MoveL Offs(p0,431.3,226.6, 0), v100, z5, tool0;
MoveL Offs(p0,430.26560000000006,226.81200000000004, 0), v100, z5, tool0;
MoveL Offs(p0,429.7934,226.93749999999994, 0), v100, z5, tool0;
MoveL Offs(p0,429.36080000000004,227.07200000000003, 0), v100, z5, tool0;
MoveL Offs(p0,428.975,227.2125, 0), v100, z5, tool0;
MoveL Offs(p0,428.6432,227.356, 0), v100, z5, tool0;
MoveL Offs(p0,428.37260000000003,227.49949999999998, 0), v100, z5, tool0;
MoveL Offs(p0,428.1704,227.64000000000001, 0), v100, z5, tool0;
MoveL Offs(p0,428.04380000000003,227.77450000000005, 0), v100, z5, tool0;
MoveL Offs(p0,428.0,227.9, 0), v100, z5, tool0;
MoveL Offs(p0,427.0009999999999,228.11059999999998, 0), v100, z5, tool0;
MoveL Offs(p0,426.27200000000005,228.15120000000002, 0), v100, z5, tool0;
MoveL Offs(p0,425.375,228.175, 0), v100, z5, tool0;
MoveL Offs(p0,424.3280000000001,228.1808, 0), v100, z5, tool0;
MoveL Offs(p0,423.149,228.1674, 0), v100, z5, tool0;
MoveL Offs(p0,421.85600000000005,228.13360000000003, 0), v100, z5, tool0;
MoveL Offs(p0,410.99179999999996,228.3078, 0), v100, z5, tool0;
MoveL Offs(p0,411.1,228.5, 0), v100, z5, tool0;
MoveL Offs(p0,411.9424000000001,228.8344000000001, 0), v100, z5, tool0;
MoveL Offs(p0,412.7326,228.9806, 0), v100, z5, tool0;
MoveL Offs(p0,413.73519999999996,229.1112, 0), v100, z5, tool0;
MoveL Offs(p0,414.925,229.225, 0), v100, z5, tool0;
MoveL Offs(p0,416.2768,229.32080000000002, 0), v100, z5, tool0;
MoveL Offs(p0,417.76540000000006,229.3974, 0), v100, z5, tool0;
MoveL Offs(p0,419.3656,229.4536, 0), v100, z5, tool0;
MoveL Offs(p0,421.0522000000001,229.4882, 0), v100, z5, tool0;
MoveL Offs(p0,422.8,229.5, 0), v100, z5, tool0;
MoveL Offs(p0,431.6752,229.20240000000004, 0), v100, z5, tool0;
MoveL Offs(p0,433.1875,228.9375, 0), v100, z5, tool0;
MoveL Offs(p0,434.63680000000005,228.5496, 0), v100, z5, tool0;
MoveL Offs(p0,436.13289999999995,228.01530000000002, 0), v100, z5, tool0;
MoveL Offs(p0,437.7856,227.3112, 0), v100, z5, tool0;
MoveL Offs(p0,439.70470000000006,226.4139, 0), v100, z5, tool0;
MoveL Offs(p0,442.0,225.3, 0), v100, z5, tool0;
MoveL Offs(p0,448.8923,221.3112, 0), v100, z5, tool0;
MoveL Offs(p0,454.77840000000015,216.69360000000006, 0), v100, z5, tool0;
MoveL Offs(p0,459.6121,211.5804, 0), v100, z5, tool0;
MoveL Offs(p0,463.34720000000004,206.1048, 0), v100, z5, tool0;
MoveL Offs(p0,465.9375,200.4, 0), v100, z5, tool0;
MoveL Offs(p0,467.33680000000004,194.5992, 0), v100, z5, tool0;
MoveL Offs(p0,467.49889999999994,188.8356, 0), v100, z5, tool0;
MoveL Offs(p0,466.3776,183.2424, 0), v100, z5, tool0;
MoveL Offs(p0,463.9267,177.9528, 0), v100, z5, tool0;
MoveL Offs(p0,460.1,173.1, 0), v100, z5, tool0;
MoveL Offs(p0,458.00750000000005,171.084, 0), v100, z5, tool0;
MoveL Offs(p0,455.96000000000004,169.34400000000005, 0), v100, z5, tool0;
MoveL Offs(p0,453.9125,167.86200000000002, 0), v100, z5, tool0;
MoveL Offs(p0,451.82000000000005,166.62000000000003, 0), v100, z5, tool0;
MoveL Offs(p0,449.6375,165.6, 0), v100, z5, tool0;
MoveL Offs(p0,447.32,164.784, 0), v100, z5, tool0;
MoveL Offs(p0,444.82250000000005,164.154, 0), v100, z5, tool0;
MoveL Offs(p0,442.1,163.692, 0), v100, z5, tool0;
MoveL Offs(p0,439.10749999999996,163.38, 0), v100, z5, tool0;
MoveL Offs(p0,435.8,163.2, 0), v100, z5, tool0;
MoveL Offs(p0,425.2664,163.5024, 0), v100, z5, tool0;
MoveL Offs(p0,423.8902,163.76069999999999, 0), v100, z5, tool0;
MoveL Offs(p0,422.50079999999997,164.0928, 0), v100, z5, tool0;
MoveL Offs(p0,421.0526,164.50410000000002, 0), v100, z5, tool0;
MoveL Offs(p0,419.5,165.0, 0), v100, z5, tool0;
MoveL Offs(p0,418.4228,165.3736, 0), v100, z5, tool0;
MoveL Offs(p0,417.36240000000015,165.76880000000003, 0), v100, z5, tool0;
MoveL Offs(p0,416.3356,166.1772, 0), v100, z5, tool0;
MoveL Offs(p0,415.3592,166.59040000000002, 0), v100, z5, tool0;
MoveL Offs(p0,414.45,167.0, 0), v100, z5, tool0;
MoveL Offs(p0,413.62479999999994,167.3976, 0), v100, z5, tool0;
MoveL Offs(p0,412.9004,167.7748, 0), v100, z5, tool0;
MoveL Offs(p0,412.2936000000001,168.12320000000003, 0), v100, z5, tool0;
MoveL Offs(p0,411.82120000000003,168.4344, 0), v100, z5, tool0;
MoveL Offs(p0,411.5,168.7, 0), v100, z5, tool0;
MoveL Offs(p0,411.22180000000014,168.9393, 0), v100, z5, tool0;
MoveL Offs(p0,410.9304000000001,169.17440000000005, 0), v100, z5, tool0;
MoveL Offs(p0,410.63059999999996,169.4011, 0), v100, z5, tool0;
MoveL Offs(p0,410.3272,169.61520000000002, 0), v100, z5, tool0;
MoveL Offs(p0,410.025,169.8125, 0), v100, z5, tool0;
MoveL Offs(p0,409.72880000000004,169.9888, 0), v100, z5, tool0;
MoveL Offs(p0,409.4434,170.13989999999998, 0), v100, z5, tool0;
MoveL Offs(p0,409.17359999999996,170.2616, 0), v100, z5, tool0;
MoveL Offs(p0,408.92420000000004,170.3497, 0), v100, z5, tool0;
MoveL Offs(p0,408.7,170.4, 0), v100, z5, tool0;
MoveL Offs(p0,407.1136000000001,170.85280000000006, 0), v100, z5, tool0;
MoveL Offs(p0,406.3384,171.20819999999998, 0), v100, z5, tool0;
MoveL Offs(p0,405.6088000000001,171.62240000000003, 0), v100, z5, tool0;
MoveL Offs(p0,404.95,172.075, 0), v100, z5, tool0;
MoveL Offs(p0,404.3872,172.54559999999998, 0), v100, z5, tool0;
MoveL Offs(p0,403.9456,173.0138, 0), v100, z5, tool0;
MoveL Offs(p0,403.65040000000005,173.4592, 0), v100, z5, tool0;
MoveL Offs(p0,403.52680000000004,173.8614, 0), v100, z5, tool0;
MoveL Offs(p0,403.6,174.2, 0), v100, z5, tool0;
MoveL Offs(p0,403.8223,174.67069999999998, 0), v100, z5, tool0;
MoveL Offs(p0,403.83360000000005,174.75840000000002, 0), v100, z5, tool0;
MoveL Offs(p0,403.8125,174.8125, 0), v100, z5, tool0;
MoveL Offs(p0,403.3921,174.7049, 0), v100, z5, tool0;
MoveL Offs(p0,403.2,174.6, 0), v100, z5, tool0;
MoveL Offs(p0,401.24240000000015,175.26400000000007, 0), v100, z5, tool0;
MoveL Offs(p0,399.7251,176.45850000000002, 0), v100, z5, tool0;
MoveL Offs(p0,397.9552,178.11200000000002, 0), v100, z5, tool0;
MoveL Offs(p0,396.0125,180.1375, 0), v100, z5, tool0;
MoveL Offs(p0,393.9768,182.448, 0), v100, z5, tool0;
MoveL Offs(p0,391.9279,184.9565, 0), v100, z5, tool0;
MoveL Offs(p0,389.94560000000007,187.57600000000002, 0), v100, z5, tool0;
MoveL Offs(p0,388.10970000000003,190.2195, 0), v100, z5, tool0;
MoveL Offs(p0,386.5,192.8, 0), v100, z5, tool0;
MoveL Offs(p0,385.22280000000006,195.07940000000002, 0), v100, z5, tool0;
MoveL Offs(p0,383.87840000000017,197.65520000000004, 0), v100, z5, tool0;
MoveL Offs(p0,382.5076,200.43380000000002, 0), v100, z5, tool0;
MoveL Offs(p0,381.1512,203.32160000000002, 0), v100, z5, tool0;
MoveL Offs(p0,379.85,206.225, 0), v100, z5, tool0;
MoveL Offs(p0,378.6448,209.05040000000002, 0), v100, z5, tool0;
MoveL Offs(p0,377.57640000000004,211.7042, 0), v100, z5, tool0;
MoveL Offs(p0,376.6856,214.09279999999998, 0), v100, z5, tool0;
MoveL Offs(p0,376.0132,216.1226, 0), v100, z5, tool0;
MoveL Offs(p0,375.6,217.7, 0), v100, z5, tool0;
MoveL Offs(p0,375.1392,219.68720000000002, 0), v100, z5, tool0;
MoveL Offs(p0,374.49360000000013,221.77760000000006, 0), v100, z5, tool0;
MoveL Offs(p0,373.6884,223.92439999999996, 0), v100, z5, tool0;
MoveL Offs(p0,372.7488000000001,226.0808, 0), v100, z5, tool0;
MoveL Offs(p0,371.7,228.2, 0), v100, z5, tool0;
MoveL Offs(p0,370.56719999999996,230.2352, 0), v100, z5, tool0;
MoveL Offs(p0,369.3756,232.13959999999997, 0), v100, z5, tool0;
MoveL Offs(p0,368.15040000000005,233.86640000000003, 0), v100, z5, tool0;
MoveL Offs(p0,366.9168,235.36880000000002, 0), v100, z5, tool0;
MoveL Offs(p0,365.7,236.6, 0), v100, z5, tool0;
MoveL Offs(p0,363.6746,238.30100000000002, 0), v100, z5, tool0;
MoveL Offs(p0,361.6168000000001,239.74400000000009, 0), v100, z5, tool0;
MoveL Offs(p0,359.52419999999995,240.929, 0), v100, z5, tool0;
MoveL Offs(p0,357.3944,241.85600000000005, 0), v100, z5, tool0;
MoveL Offs(p0,355.225,242.525, 0), v100, z5, tool0;
MoveL Offs(p0,353.0136,242.93599999999998, 0), v100, z5, tool0;
MoveL Offs(p0,350.75780000000003,243.08900000000003, 0), v100, z5, tool0;
MoveL Offs(p0,348.45520000000005,242.984, 0), v100, z5, tool0;
MoveL Offs(p0,346.1034,242.621, 0), v100, z5, tool0;
MoveL Offs(p0,343.7,242.0, 0), v100, z5, tool0;
MoveL Offs(p0,338.0,240.2, 0), v100, z5, tool0;
MoveL Offs(p0,338.0,243.0, 0), v100, z5, tool0;
MoveL Offs(p0,338.43520000000007,245.01520000000005, 0), v100, z5, tool0;
MoveL Offs(p0,339.0098,245.79179999999997, 0), v100, z5, tool0;
MoveL Offs(p0,339.84959999999995,246.42560000000003, 0), v100, z5, tool0;
MoveL Offs(p0,340.975,246.925, 0), v100, z5, tool0;
MoveL Offs(p0,342.40639999999996,247.2984, 0), v100, z5, tool0;
MoveL Offs(p0,344.1642,247.55419999999998, 0), v100, z5, tool0;
MoveL Offs(p0,346.2688,247.70080000000002, 0), v100, z5, tool0;
MoveL Offs(p0,348.7406,247.7466, 0), v100, z5, tool0;
MoveL Offs(p0,351.6,247.7, 0), v100, z5, tool0;
MoveL Offs(p0,355.35920000000004,247.4872000000001, 0), v100, z5, tool0;
MoveL Offs(p0,356.85779999999994,247.3328, 0), v100, z5, tool0;
MoveL Offs(p0,358.17760000000004,247.1256, 0), v100, z5, tool0;
MoveL Offs(p0,359.375,246.85, 0), v100, z5, tool0;
MoveL Offs(p0,360.50640000000004,246.4904, 0), v100, z5, tool0;
MoveL Offs(p0,361.6282,246.03119999999998, 0), v100, z5, tool0;
MoveL Offs(p0,362.79679999999996,245.45680000000002, 0), v100, z5, tool0;
MoveL Offs(p0,364.0686,244.7516, 0), v100, z5, tool0;
MoveL Offs(p0,365.5,243.9, 0), v100, z5, tool0;
MoveL Offs(p0,365.5,243.9, 0), v100, z5, tool0;
MoveJ Offs(p0,333.7,242.7, 10), v100, z1, tool0;
MoveL Offs(p0,333.3992,241.44880000000003, 0), v100, z5, tool0;
MoveL Offs(p0,333.2194,241.6821, 0), v100, z5, tool0;
MoveL Offs(p0,333.0,242.0, 0), v100, z5, tool0;
MoveL Offs(p0,332.6946000000001,242.54360000000003, 0), v100, z5, tool0;
MoveL Offs(p0,332.44080000000014,243.13280000000003, 0), v100, z5, tool0;
MoveL Offs(p0,332.2422,243.7352, 0), v100, z5, tool0;
MoveL Offs(p0,332.10240000000005,244.31840000000003, 0), v100, z5, tool0;
MoveL Offs(p0,332.025,244.85, 0), v100, z5, tool0;
MoveL Offs(p0,332.0136,245.29759999999996, 0), v100, z5, tool0;
MoveL Offs(p0,332.0718,245.6288, 0), v100, z5, tool0;
MoveL Offs(p0,332.20320000000004,245.8112, 0), v100, z5, tool0;
MoveL Offs(p0,332.4114,245.81239999999997, 0), v100, z5, tool0;
MoveL Offs(p0,332.7,245.6, 0), v100, z5, tool0;
MoveL Offs(p0,332.9384000000001,245.29840000000007, 0), v100, z5, tool0;
MoveL Offs(p0,333.0546,245.06809999999996, 0), v100, z5, tool0;
MoveL Offs(p0,333.16720000000004,244.79520000000002, 0), v100, z5, tool0;
MoveL Offs(p0,333.275,244.4875, 0), v100, z5, tool0;
MoveL Offs(p0,333.3768,244.15279999999998, 0), v100, z5, tool0;
MoveL Offs(p0,333.4714,243.7989, 0), v100, z5, tool0;
MoveL Offs(p0,333.5576,243.4336, 0), v100, z5, tool0;
MoveL Offs(p0,333.6342,243.0647, 0), v100, z5, tool0;
MoveL Offs(p0,333.7,242.7, 0), v100, z5, tool0;
MoveL Offs(p0,333.7,242.7, 0), v100, z5, tool0;
MoveJ Offs(p0,201.3,238.9, 10), v100, z1, tool0;
MoveL Offs(p0,202.17000000000002,238.3953, 0), v100, z5, tool0;
MoveL Offs(p0,203.13600000000005,237.74240000000003, 0), v100, z5, tool0;
MoveL Offs(p0,204.16199999999998,236.9731, 0), v100, z5, tool0;
MoveL Offs(p0,205.212,236.11920000000003, 0), v100, z5, tool0;
MoveL Offs(p0,206.25,235.2125, 0), v100, z5, tool0;
MoveL Offs(p0,207.24,234.2848, 0), v100, z5, tool0;
MoveL Offs(p0,208.14600000000002,233.36790000000002, 0), v100, z5, tool0;
MoveL Offs(p0,208.93200000000002,232.49360000000001, 0), v100, z5, tool0;
MoveL Offs(p0,209.56199999999998,231.69369999999998, 0), v100, z5, tool0;
MoveL Offs(p0,210.0,231.0, 0), v100, z5, tool0;
MoveL Offs(p0,209.68800000000002,229.92960000000002, 0), v100, z5, tool0;
MoveL Offs(p0,209.1375,229.8, 0), v100, z5, tool0;
MoveL Offs(p0,208.344,229.71840000000003, 0), v100, z5, tool0;
MoveL Offs(p0,207.2805,229.6812, 0), v100, z5, tool0;
MoveL Offs(p0,205.92000000000002,229.6848, 0), v100, z5, tool0;
MoveL Offs(p0,204.2355,229.72560000000004, 0), v100, z5, tool0;
MoveL Offs(p0,202.2,229.8, 0), v100, z5, tool0;
MoveL Offs(p0,188.76839999999999,229.2276, 0), v100, z5, tool0;
MoveL Offs(p0,183.70880000000002,228.5232, 0), v100, z5, tool0;
MoveL Offs(p0,178.3,227.55, 0), v100, z5, tool0;
MoveL Offs(p0,172.50719999999995,226.30079999999998, 0), v100, z5, tool0;
MoveL Offs(p0,166.2956,224.76839999999999, 0), v100, z5, tool0;
MoveL Offs(p0,159.6304,222.9456, 0), v100, z5, tool0;
MoveL Offs(p0,152.4768,220.8252, 0), v100, z5, tool0;
MoveL Offs(p0,144.8,218.4, 0), v100, z5, tool0;
MoveL Offs(p0,137.62550000000002,215.98860000000005, 0), v100, z5, tool0;
MoveL Offs(p0,130.28000000000003,213.31680000000006, 0), v100, z5, tool0;
MoveL Offs(p0,122.97050000000002,210.47819999999996, 0), v100, z5, tool0;
MoveL Offs(p0,115.90400000000002,207.56640000000002, 0), v100, z5, tool0;
MoveL Offs(p0,109.2875,204.675, 0), v100, z5, tool0;
MoveL Offs(p0,103.328,201.8976, 0), v100, z5, tool0;
MoveL Offs(p0,98.23249999999999,199.3278, 0), v100, z5, tool0;
MoveL Offs(p0,94.20800000000001,197.0592, 0), v100, z5, tool0;
MoveL Offs(p0,91.4615,195.18540000000002, 0), v100, z5, tool0;
MoveL Offs(p0,90.2,193.8, 0), v100, z5, tool0;
MoveL Offs(p0,89.98890000000002,193.48160000000001, 0), v100, z5, tool0;
MoveL Offs(p0,89.67520000000002,193.24480000000003, 0), v100, z5, tool0;
MoveL Offs(p0,89.2883,193.0872, 0), v100, z5, tool0;
MoveL Offs(p0,88.85760000000002,193.0064, 0), v100, z5, tool0;
MoveL Offs(p0,88.4125,193.0, 0), v100, z5, tool0;
MoveL Offs(p0,87.9824,193.0656, 0), v100, z5, tool0;
MoveL Offs(p0,87.5967,193.2008, 0), v100, z5, tool0;
MoveL Offs(p0,87.2848,193.40320000000003, 0), v100, z5, tool0;
MoveL Offs(p0,87.0,194.0, 0), v100, z5, tool0;
MoveL Offs(p0,86.7376,194.6112, 0), v100, z5, tool0;
MoveL Offs(p0,86.6,194.725, 0), v100, z5, tool0;
MoveL Offs(p0,86.43839999999999,194.82080000000002, 0), v100, z5, tool0;
MoveL Offs(p0,86.2552,194.8974, 0), v100, z5, tool0;
MoveL Offs(p0,86.0528,194.9536, 0), v100, z5, tool0;
MoveL Offs(p0,85.8336,194.9882, 0), v100, z5, tool0;
MoveL Offs(p0,85.6,195.0, 0), v100, z5, tool0;
MoveL Offs(p0,84.32000000000002,195.36960000000002, 0), v100, z5, tool0;
MoveL Offs(p0,83.8945,195.78839999999997, 0), v100, z5, tool0;
MoveL Offs(p0,83.61600000000001,196.3248, 0), v100, z5, tool0;
MoveL Offs(p0,83.4875,196.95, 0), v100, z5, tool0;
MoveL Offs(p0,83.51200000000001,197.6352, 0), v100, z5, tool0;
MoveL Offs(p0,83.6925,198.35160000000002, 0), v100, z5, tool0;
MoveL Offs(p0,84.03200000000001,199.0704, 0), v100, z5, tool0;
MoveL Offs(p0,84.5335,199.76280000000003, 0), v100, z5, tool0;
MoveL Offs(p0,85.2,200.4, 0), v100, z5, tool0;
MoveL Offs(p0,86.3957,201.25300000000001, 0), v100, z5, tool0;
MoveL Offs(p0,88.03360000000004,202.26800000000006, 0), v100, z5, tool0;
MoveL Offs(p0,89.9799,203.379, 0), v100, z5, tool0;
MoveL Offs(p0,92.10080000000002,204.52000000000004, 0), v100, z5, tool0;
MoveL Offs(p0,94.2625,205.625, 0), v100, z5, tool0;
MoveL Offs(p0,96.3312,206.62800000000001, 0), v100, z5, tool0;
MoveL Offs(p0,98.1731,207.46300000000002, 0), v100, z5, tool0;
MoveL Offs(p0,99.65440000000001,208.06400000000002, 0), v100, z5, tool0;
MoveL Offs(p0,100.6413,208.365, 0), v100, z5, tool0;
MoveL Offs(p0,101.0,208.3, 0), v100, z5, tool0;
MoveL Offs(p0,101.25,208.0375, 0), v100, z5, tool0;
MoveL Offs(p0,101.3456,208.09120000000001, 0), v100, z5, tool0;
MoveL Offs(p0,101.8,208.6, 0), v100, z5, tool0;
MoveL Offs(p0,102.76490000000001,209.33620000000005, 0), v100, z5, tool0;
MoveL Offs(p0,104.76720000000003,210.39760000000007, 0), v100, z5, tool0;
MoveL Offs(p0,107.5483,211.68339999999998, 0), v100, z5, tool0;
MoveL Offs(p0,110.84960000000001,213.09280000000004, 0), v100, z5, tool0;
MoveL Offs(p0,114.4125,214.525, 0), v100, z5, tool0;
MoveL Offs(p0,117.97840000000001,215.87920000000003, 0), v100, z5, tool0;
MoveL Offs(p0,121.28870000000002,217.05460000000002, 0), v100, z5, tool0;
MoveL Offs(p0,124.08480000000002,217.9504, 0), v100, z5, tool0;
MoveL Offs(p0,126.10810000000001,218.46580000000003, 0), v100, z5, tool0;
MoveL Offs(p0,127.1,218.5, 0), v100, z5, tool0;
MoveL Offs(p0,127.46960000000004,218.27120000000008, 0), v100, z5, tool0;
MoveL Offs(p0,127.61389999999999,218.20929999999998, 0), v100, z5, tool0;
MoveL Offs(p0,127.72880000000002,218.18159999999997, 0), v100, z5, tool0;
MoveL Offs(p0,127.8125,218.1875, 0), v100, z5, tool0;
MoveL Offs(p0,127.86319999999998,218.2264, 0), v100, z5, tool0;
MoveL Offs(p0,127.87910000000002,218.2977, 0), v100, z5, tool0;
MoveL Offs(p0,127.7,218.7, 0), v100, z5, tool0;
MoveL Offs(p0,128.13320000000002,219.17020000000002, 0), v100, z5, tool0;
MoveL Offs(p0,129.6896,220.0016000000001, 0), v100, z5, tool0;
MoveL Offs(p0,132.2144,221.13539999999998, 0), v100, z5, tool0;
MoveL Offs(p0,135.5528,222.51280000000003, 0), v100, z5, tool0;
MoveL Offs(p0,139.55,224.075, 0), v100, z5, tool0;
MoveL Offs(p0,144.05120000000002,225.7632, 0), v100, z5, tool0;
MoveL Offs(p0,148.9016,227.51859999999996, 0), v100, z5, tool0;
MoveL Offs(p0,153.9464,229.2824, 0), v100, z5, tool0;
MoveL Offs(p0,159.0308,230.9958, 0), v100, z5, tool0;
MoveL Offs(p0,164.0,232.6, 0), v100, z5, tool0;
MoveL Offs(p0,170.2905,234.5179, 0), v100, z5, tool0;
MoveL Offs(p0,175.92400000000006,236.13520000000008, 0), v100, z5, tool0;
MoveL Offs(p0,180.9335,237.45729999999998, 0), v100, z5, tool0;
MoveL Offs(p0,185.35200000000003,238.48960000000002, 0), v100, z5, tool0;
MoveL Offs(p0,189.2125,239.2375, 0), v100, z5, tool0;
MoveL Offs(p0,192.548,239.70639999999997, 0), v100, z5, tool0;
MoveL Offs(p0,195.3915,239.90169999999998, 0), v100, z5, tool0;
MoveL Offs(p0,197.776,239.82880000000006, 0), v100, z5, tool0;
MoveL Offs(p0,199.7345,239.4931, 0), v100, z5, tool0;
MoveL Offs(p0,201.3,238.9, 0), v100, z5, tool0;
MoveL Offs(p0,201.3,238.9, 0), v100, z5, tool0;
MoveJ Offs(p0,169.0,237.4, 10), v100, z1, tool0;
MoveL Offs(p0,168.7024,237.1728, 0), v100, z5, tool0;
MoveL Offs(p0,168.55,237.125, 0), v100, z5, tool0;
MoveL Offs(p0,168.37359999999998,237.08319999999998, 0), v100, z5, tool0;
MoveL Offs(p0,168.17680000000001,237.0486, 0), v100, z5, tool0;
MoveL Offs(p0,167.9632,237.0224, 0), v100, z5, tool0;
MoveL Offs(p0,167.7364,237.0058, 0), v100, z5, tool0;
MoveL Offs(p0,167.5,237.0, 0), v100, z5, tool0;
MoveL Offs(p0,166.45,237.275, 0), v100, z5, tool0;
MoveL Offs(p0,166.2976,237.3888, 0), v100, z5, tool0;
MoveL Offs(p0,166.1728,237.5194, 0), v100, z5, tool0;
MoveL Offs(p0,166.07920000000001,237.66559999999998, 0), v100, z5, tool0;
MoveL Offs(p0,166.0204,237.82620000000003, 0), v100, z5, tool0;
MoveL Offs(p0,166.0,238.0, 0), v100, z5, tool0;
MoveL Offs(p0,166.29760000000002,238.44320000000002, 0), v100, z5, tool0;
MoveL Offs(p0,166.45,238.5, 0), v100, z5, tool0;
MoveL Offs(p0,166.62640000000002,238.5328, 0), v100, z5, tool0;
MoveL Offs(p0,166.82319999999999,238.54039999999995, 0), v100, z5, tool0;
MoveL Offs(p0,167.03680000000003,238.52160000000003, 0), v100, z5, tool0;
MoveL Offs(p0,167.2636,238.4752, 0), v100, z5, tool0;
MoveL Offs(p0,167.5,238.4, 0), v100, z5, tool0;
MoveL Offs(p0,167.96320000000003,238.16160000000008, 0), v100, z5, tool0;
MoveL Offs(p0,168.17680000000001,238.04539999999997, 0), v100, z5, tool0;
MoveL Offs(p0,168.3736,237.93280000000004, 0), v100, z5, tool0;
MoveL Offs(p0,168.55,237.825, 0), v100, z5, tool0;
MoveL Offs(p0,168.7024,237.7232, 0), v100, z5, tool0;
MoveL Offs(p0,168.8272,237.6286, 0), v100, z5, tool0;
MoveL Offs(p0,168.9208,237.5424, 0), v100, z5, tool0;
MoveL Offs(p0,168.97960000000003,237.46580000000003, 0), v100, z5, tool0;
MoveL Offs(p0,169.0,237.4, 0), v100, z5, tool0;
MoveL Offs(p0,169.0,237.4, 0), v100, z5, tool0;
MoveJ Offs(p0,48.2,226.6, 10), v100, z1, tool0;
MoveL Offs(p0,51.083000000000006,225.5016, 0), v100, z5, tool0;
MoveL Offs(p0,53.55200000000001,224.12480000000005, 0), v100, z5, tool0;
MoveL Offs(p0,55.607000000000006,222.46719999999996, 0), v100, z5, tool0;
MoveL Offs(p0,57.248000000000005,220.52639999999997, 0), v100, z5, tool0;
MoveL Offs(p0,58.475,218.3, 0), v100, z5, tool0;
MoveL Offs(p0,59.28800000000001,215.7856, 0), v100, z5, tool0;
MoveL Offs(p0,59.687,212.9808, 0), v100, z5, tool0;
MoveL Offs(p0,59.672000000000004,209.88320000000004, 0), v100, z5, tool0;
MoveL Offs(p0,59.24300000000001,206.4904, 0), v100, z5, tool0;
MoveL Offs(p0,58.4,202.8, 0), v100, z5, tool0;
MoveL Offs(p0,58.19,201.4805, 0), v100, z5, tool0;
MoveL Offs(p0,58.16000000000001,201.28000000000003, 0), v100, z5, tool0;
MoveL Offs(p0,58.129999999999995,201.0855, 0), v100, z5, tool0;
MoveL Offs(p0,58.1,200.9, 0), v100, z5, tool0;
MoveL Offs(p0,57.8856,200.4568, 0), v100, z5, tool0;
MoveL Offs(p0,57.775,200.4, 0), v100, z5, tool0;
MoveL Offs(p0,57.64639999999999,200.36719999999997, 0), v100, z5, tool0;
MoveL Offs(p0,57.502199999999995,200.3596, 0), v100, z5, tool0;
MoveL Offs(p0,57.344800000000006,200.3784, 0), v100, z5, tool0;
MoveL Offs(p0,57.17660000000001,200.4248, 0), v100, z5, tool0;
MoveL Offs(p0,57.0,200.5, 0), v100, z5, tool0;
MoveL Offs(p0,56.4596,200.248, 0), v100, z5, tool0;
MoveL Offs(p0,56.47840000000001,200.06800000000004, 0), v100, z5, tool0;
MoveL Offs(p0,56.524800000000006,199.85200000000003, 0), v100, z5, tool0;
MoveL Offs(p0,56.6,199.6, 0), v100, z5, tool0;
MoveL Offs(p0,56.2193,196.98549999999997, 0), v100, z5, tool0;
MoveL Offs(p0,55.76160000000001,195.76000000000002, 0), v100, z5, tool0;
MoveL Offs(p0,55.1875,194.4625, 0), v100, z5, tool0;
MoveL Offs(p0,54.52639999999999,193.156, 0), v100, z5, tool0;
MoveL Offs(p0,53.8077,191.90350000000004, 0), v100, z5, tool0;
MoveL Offs(p0,53.06080000000001,190.76800000000003, 0), v100, z5, tool0;
MoveL Offs(p0,52.31510000000001,189.8125, 0), v100, z5, tool0;
MoveL Offs(p0,51.6,189.1, 0), v100, z5, tool0;
MoveL Offs(p0,51.2356,188.80980000000005, 0), v100, z5, tool0;
MoveL Offs(p0,50.916800000000016,188.60240000000005, 0), v100, z5, tool0;
MoveL Offs(p0,50.6352,188.4826, 0), v100, z5, tool0;
MoveL Offs(p0,50.382400000000004,188.45520000000002, 0), v100, z5, tool0;
MoveL Offs(p0,50.15,188.525, 0), v100, z5, tool0;
MoveL Offs(p0,49.92959999999999,188.6968, 0), v100, z5, tool0;
MoveL Offs(p0,49.491200000000006,189.36560000000003, 0), v100, z5, tool0;
MoveL Offs(p0,49.2564,189.8722, 0), v100, z5, tool0;
MoveL Offs(p0,49.0,190.5, 0), v100, z5, tool0;
MoveL Offs(p0,48.689600000000006,191.40240000000003, 0), v100, z5, tool0;
MoveL Offs(p0,48.5734,191.84459999999996, 0), v100, z5, tool0;
MoveL Offs(p0,48.4848,192.27120000000002, 0), v100, z5, tool0;
MoveL Offs(p0,48.425,192.675, 0), v100, z5, tool0;
MoveL Offs(p0,48.3952,193.04879999999997, 0), v100, z5, tool0;
MoveL Offs(p0,48.3966,193.38539999999998, 0), v100, z5, tool0;
MoveL Offs(p0,48.430400000000006,193.67760000000004, 0), v100, z5, tool0;
MoveL Offs(p0,48.4978,193.9182, 0), v100, z5, tool0;
MoveL Offs(p0,48.6,194.1, 0), v100, z5, tool0;
MoveL Offs(p0,48.3,194.8, 0), v100, z5, tool0;
MoveL Offs(p0,47.333600000000004,195.12640000000002, 0), v100, z5, tool0;
MoveL Offs(p0,46.975,195.3625, 0), v100, z5, tool0;
MoveL Offs(p0,46.5864,195.64960000000002, 0), v100, z5, tool0;
MoveL Offs(p0,46.176199999999994,195.98229999999998, 0), v100, z5, tool0;
MoveL Offs(p0,45.7528,196.35520000000002, 0), v100, z5, tool0;
MoveL Offs(p0,45.3246,196.7629, 0), v100, z5, tool0;
MoveL Offs(p0,44.9,197.2, 0), v100, z5, tool0;
MoveL Offs(p0,43.92960000000001,198.06340000000003, 0), v100, z5, tool0;
MoveL Offs(p0,42.82480000000001,198.85120000000006, 0), v100, z5, tool0;
MoveL Offs(p0,41.59519999999999,199.5598, 0), v100, z5, tool0;
MoveL Offs(p0,40.2504,200.1856, 0), v100, z5, tool0;
MoveL Offs(p0,38.8,200.725, 0), v100, z5, tool0;
MoveL Offs(p0,37.2536,201.1744, 0), v100, z5, tool0;
MoveL Offs(p0,35.620799999999996,201.53019999999998, 0), v100, z5, tool0;
MoveL Offs(p0,33.911199999999994,201.7888, 0), v100, z5, tool0;
MoveL Offs(p0,32.13440000000001,201.94660000000002, 0), v100, z5, tool0;
MoveL Offs(p0,30.3,202.0, 0), v100, z5, tool0;
MoveL Offs(p0,26.2,202.0, 0), v100, z5, tool0;
MoveL Offs(p0,28.1,208.3, 0), v100, z5, tool0;
MoveL Offs(p0,28.396200000000004,209.35530000000003, 0), v100, z5, tool0;
MoveL Offs(p0,28.681600000000003,210.46640000000008, 0), v100, z5, tool0;
MoveL Offs(p0,28.9514,211.6111, 0), v100, z5, tool0;
MoveL Offs(p0,29.200799999999997,212.7672, 0), v100, z5, tool0;
MoveL Offs(p0,29.425,213.9125, 0), v100, z5, tool0;
MoveL Offs(p0,29.6192,215.0248, 0), v100, z5, tool0;
MoveL Offs(p0,29.7786,216.0819, 0), v100, z5, tool0;
MoveL Offs(p0,29.898400000000002,217.0616, 0), v100, z5, tool0;
MoveL Offs(p0,29.9738,217.9417, 0), v100, z5, tool0;
MoveL Offs(p0,30.0,218.7, 0), v100, z5, tool0;
MoveL Offs(p0,30.352000000000004,222.07280000000006, 0), v100, z5, tool0;
MoveL Offs(p0,30.6125,222.6625, 0), v100, z5, tool0;
MoveL Offs(p0,30.972,223.2072, 0), v100, z5, tool0;
MoveL Offs(p0,31.4455,223.73509999999996, 0), v100, z5, tool0;
MoveL Offs(p0,32.048,224.27439999999996, 0), v100, z5, tool0;
MoveL Offs(p0,32.7945,224.85330000000005, 0), v100, z5, tool0;
MoveL Offs(p0,33.7,225.5, 0), v100, z5, tool0;
MoveL Offs(p0,34.96730000000001,226.26520000000005, 0), v100, z5, tool0;
MoveL Offs(p0,36.20640000000001,226.88160000000008, 0), v100, z5, tool0;
MoveL Offs(p0,37.4431,227.35040000000004, 0), v100, z5, tool0;
MoveL Offs(p0,38.7032,227.6728, 0), v100, z5, tool0;
MoveL Offs(p0,40.0125,227.85, 0), v100, z5, tool0;
MoveL Offs(p0,41.3968,227.8832, 0), v100, z5, tool0;
MoveL Offs(p0,42.881899999999995,227.7736, 0), v100, z5, tool0;
MoveL Offs(p0,44.4936,227.5224, 0), v100, z5, tool0;
MoveL Offs(p0,46.2577,227.1308, 0), v100, z5, tool0;
MoveL Offs(p0,48.2,226.6, 0), v100, z5, tool0;
MoveL Offs(p0,48.2,226.6, 0), v100, z5, tool0;
MoveJ Offs(p0,209.9,227.4, 10), v100, z1, tool0;
MoveL Offs(p0,211.07630000000003,227.07440000000005, 0), v100, z5, tool0;
MoveL Offs(p0,211.96640000000002,226.64320000000006, 0), v100, z5, tool0;
MoveL Offs(p0,212.5721,226.11479999999997, 0), v100, z5, tool0;
MoveL Offs(p0,212.89520000000002,225.4976, 0), v100, z5, tool0;
MoveL Offs(p0,212.9375,224.8, 0), v100, z5, tool0;
MoveL Offs(p0,212.7008,224.03040000000001, 0), v100, z5, tool0;
MoveL Offs(p0,212.18689999999998,223.19719999999998, 0), v100, z5, tool0;
MoveL Offs(p0,211.3976,222.30880000000002, 0), v100, z5, tool0;
MoveL Offs(p0,210.33469999999997,221.37359999999998, 0), v100, z5, tool0;
MoveL Offs(p0,209.0,220.4, 0), v100, z5, tool0;
MoveL Offs(p0,207.7799,219.58109999999996, 0), v100, z5, tool0;
MoveL Offs(p0,206.8112,218.90080000000006, 0), v100, z5, tool0;
MoveL Offs(p0,206.08129999999997,218.32369999999997, 0), v100, z5, tool0;
MoveL Offs(p0,205.57760000000002,217.81440000000003, 0), v100, z5, tool0;
MoveL Offs(p0,205.2875,217.3375, 0), v100, z5, tool0;
MoveL Offs(p0,205.1984,216.8576, 0), v100, z5, tool0;
MoveL Offs(p0,205.2977,216.3393, 0), v100, z5, tool0;
MoveL Offs(p0,205.5728,215.74720000000002, 0), v100, z5, tool0;
MoveL Offs(p0,206.01110000000003,215.0459, 0), v100, z5, tool0;
MoveL Offs(p0,206.6,214.2, 0), v100, z5, tool0;
MoveL Offs(p0,206.92690000000002,213.69790000000006, 0), v100, z5, tool0;
MoveL Offs(p0,207.18720000000002,213.26720000000006, 0), v100, z5, tool0;
MoveL Offs(p0,207.38029999999998,212.9013, 0), v100, z5, tool0;
MoveL Offs(p0,207.50560000000002,212.5936, 0), v100, z5, tool0;
MoveL Offs(p0,207.5625,212.3375, 0), v100, z5, tool0;
MoveL Offs(p0,207.5504,212.12639999999996, 0), v100, z5, tool0;
MoveL Offs(p0,207.46869999999998,211.95369999999997, 0), v100, z5, tool0;
MoveL Offs(p0,207.3168,211.8128, 0), v100, z5, tool0;
MoveL Offs(p0,207.09409999999997,211.69710000000003, 0), v100, z5, tool0;
MoveL Offs(p0,206.8,211.6, 0), v100, z5, tool0;
MoveL Offs(p0,199.7811,209.37510000000006, 0), v100, z5, tool0;
MoveL Offs(p0,193.03280000000004,206.91680000000005, 0), v100, z5, tool0;
MoveL Offs(p0,186.5977,204.2497, 0), v100, z5, tool0;
MoveL Offs(p0,180.5184,201.3984, 0), v100, z5, tool0;
MoveL Offs(p0,174.8375,198.3875, 0), v100, z5, tool0;
MoveL Offs(p0,169.5976,195.2416, 0), v100, z5, tool0;
MoveL Offs(p0,164.8413,191.9853, 0), v100, z5, tool0;
MoveL Offs(p0,160.6112,188.64320000000004, 0), v100, z5, tool0;
MoveL Offs(p0,156.94989999999999,185.23989999999998, 0), v100, z5, tool0;
MoveL Offs(p0,153.9,181.8, 0), v100, z5, tool0;
MoveL Offs(p0,152.2259,179.5903, 0), v100, z5, tool0;
MoveL Offs(p0,151.03120000000004,177.82640000000004, 0), v100, z5, tool0;
MoveL Offs(p0,150.2973,176.5161, 0), v100, z5, tool0;
MoveL Offs(p0,150.00560000000002,175.6672, 0), v100, z5, tool0;
MoveL Offs(p0,150.1375,175.2875, 0), v100, z5, tool0;
MoveL Offs(p0,150.6744,175.38479999999998, 0), v100, z5, tool0;
MoveL Offs(p0,151.59769999999997,175.9669, 0), v100, z5, tool0;
MoveL Offs(p0,152.8888,177.04160000000002, 0), v100, z5, tool0;
MoveL Offs(p0,154.52910000000003,178.61669999999998, 0), v100, z5, tool0;
MoveL Offs(p0,156.5,180.7, 0), v100, z5, tool0;
MoveL Offs(p0,157.65310000000005,181.9107, 0), v100, z5, tool0;
MoveL Offs(p0,158.93280000000004,183.18560000000005, 0), v100, z5, tool0;
MoveL Offs(p0,160.30969999999996,184.4989, 0), v100, z5, tool0;
MoveL Offs(p0,161.7544,185.82480000000004, 0), v100, z5, tool0;
MoveL Offs(p0,163.2375,187.1375, 0), v100, z5, tool0;
MoveL Offs(p0,164.72959999999998,188.4112, 0), v100, z5, tool0;
MoveL Offs(p0,166.2013,189.6201, 0), v100, z5, tool0;
MoveL Offs(p0,167.6232,190.7384, 0), v100, z5, tool0;
MoveL Offs(p0,168.9659,191.7403, 0), v100, z5, tool0;
MoveL Offs(p0,170.2,192.6, 0), v100, z5, tool0;
MoveL Offs(p0,172.84720000000002,194.2377, 0), v100, z5, tool0;
MoveL Offs(p0,175.87360000000007,195.94560000000004, 0), v100, z5, tool0;
MoveL Offs(p0,179.1964,197.6859, 0), v100, z5, tool0;
MoveL Offs(p0,182.7328,199.4208, 0), v100, z5, tool0;
MoveL Offs(p0,186.4,201.1125, 0), v100, z5, tool0;
MoveL Offs(p0,190.11520000000002,202.7232, 0), v100, z5, tool0;
MoveL Offs(p0,193.7956,204.21509999999998, 0), v100, z5, tool0;
MoveL Offs(p0,197.35840000000002,205.55040000000002, 0), v100, z5, tool0;
MoveL Offs(p0,200.7208,206.6913, 0), v100, z5, tool0;
MoveL Offs(p0,203.8,207.6, 0), v100, z5, tool0;
MoveL Offs(p0,205.421,208.03210000000004, 0), v100, z5, tool0;
MoveL Offs(p0,206.77200000000008,208.36880000000005, 0), v100, z5, tool0;
MoveL Offs(p0,207.89500000000004,208.6107, 0), v100, z5, tool0;
MoveL Offs(p0,208.83200000000002,208.75840000000002, 0), v100, z5, tool0;
MoveL Offs(p0,209.625,208.8125, 0), v100, z5, tool0;
MoveL Offs(p0,210.31599999999997,208.7736, 0), v100, z5, tool0;
MoveL Offs(p0,210.94700000000003,208.64229999999998, 0), v100, z5, tool0;
MoveL Offs(p0,211.56000000000003,208.4192, 0), v100, z5, tool0;
MoveL Offs(p0,212.19700000000003,208.1049, 0), v100, z5, tool0;
MoveL Offs(p0,213.60729999999998,207.29550000000003, 0), v100, z5, tool0;
MoveL Offs(p0,214.26240000000007,206.98400000000007, 0), v100, z5, tool0;
MoveL Offs(p0,214.9151,206.7685, 0), v100, z5, tool0;
MoveL Offs(p0,215.61520000000002,206.65200000000004, 0), v100, z5, tool0;
MoveL Offs(p0,216.4125,206.6375, 0), v100, z5, tool0;
MoveL Offs(p0,217.35679999999996,206.72799999999998, 0), v100, z5, tool0;
MoveL Offs(p0,218.4979,206.92649999999998, 0), v100, z5, tool0;
MoveL Offs(p0,219.8856,207.23600000000002, 0), v100, z5, tool0;
MoveL Offs(p0,223.6,208.2, 0), v100, z5, tool0;
MoveL Offs(p0,226.21560000000005,208.7911, 0), v100, z5, tool0;
MoveL Offs(p0,228.87680000000006,209.24480000000003, 0), v100, z5, tool0;
MoveL Offs(p0,231.54520000000002,209.56169999999997, 0), v100, z5, tool0;
MoveL Offs(p0,234.1824,209.7424, 0), v100, z5, tool0;
MoveL Offs(p0,236.75,209.7875, 0), v100, z5, tool0;
MoveL Offs(p0,239.2096,209.69760000000002, 0), v100, z5, tool0;
MoveL Offs(p0,241.52280000000002,209.47329999999997, 0), v100, z5, tool0;
MoveL Offs(p0,243.65120000000002,209.11520000000002, 0), v100, z5, tool0;
MoveL Offs(p0,245.55640000000002,208.6239, 0), v100, z5, tool0;
MoveL Offs(p0,247.2,208.0, 0), v100, z5, tool0;
MoveL Offs(p0,249.9,206.7, 0), v100, z5, tool0;
MoveL Offs(p0,245.5,203.8, 0), v100, z5, tool0;
MoveL Offs(p0,243.20880000000002,202.11210000000003, 0), v100, z5, tool0;
MoveL Offs(p0,240.8384000000001,200.05280000000008, 0), v100, z5, tool0;
MoveL Offs(p0,238.39359999999996,197.62869999999998, 0), v100, z5, tool0;
MoveL Offs(p0,235.8792,194.84640000000005, 0), v100, z5, tool0;
MoveL Offs(p0,233.3,191.7125, 0), v100, z5, tool0;
MoveL Offs(p0,230.66080000000002,188.23359999999997, 0), v100, z5, tool0;
MoveL Offs(p0,227.96639999999996,184.4163, 0), v100, z5, tool0;
MoveL Offs(p0,225.22160000000002,180.2672, 0), v100, z5, tool0;
MoveL Offs(p0,222.4312,175.7929, 0), v100, z5, tool0;
MoveL Offs(p0,219.6,171.0, 0), v100, z5, tool0;
MoveL Offs(p0,218.41240000000008,168.95710000000003, 0), v100, z5, tool0;
MoveL Offs(p0,217.3592000000001,167.19680000000002, 0), v100, z5, tool0;
MoveL Offs(p0,216.4248,165.70170000000002, 0), v100, z5, tool0;
MoveL Offs(p0,215.5936,164.45440000000002, 0), v100, z5, tool0;
MoveL Offs(p0,214.85,163.4375, 0), v100, z5, tool0;
MoveL Offs(p0,214.1784,162.6336, 0), v100, z5, tool0;
MoveL Offs(p0,213.5632,162.0253, 0), v100, z5, tool0;
MoveL Offs(p0,212.98880000000003,161.59520000000003, 0), v100, z5, tool0;
MoveL Offs(p0,212.4396,161.3259, 0), v100, z5, tool0;
MoveL Offs(p0,211.9,161.2, 0), v100, z5, tool0;
MoveL Offs(p0,209.68720000000008,161.4096, 0), v100, z5, tool0;
MoveL Offs(p0,208.49979999999996,161.8174, 0), v100, z5, tool0;
MoveL Offs(p0,207.3016,162.39679999999998, 0), v100, z5, tool0;
MoveL Offs(p0,206.125,163.125, 0), v100, z5, tool0;
MoveL Offs(p0,205.0024,163.9792, 0), v100, z5, tool0;
MoveL Offs(p0,203.9662,164.9366, 0), v100, z5, tool0;
MoveL Offs(p0,203.0488,165.9744, 0), v100, z5, tool0;
MoveL Offs(p0,202.2826,167.06980000000001, 0), v100, z5, tool0;
MoveL Offs(p0,201.7,168.2, 0), v100, z5, tool0;
MoveL Offs(p0,200.63980000000004,170.23610000000002, 0), v100, z5, tool0;
MoveL Offs(p0,199.32640000000006,172.08080000000004, 0), v100, z5, tool0;
MoveL Offs(p0,197.7706,173.72869999999998, 0), v100, z5, tool0;
MoveL Offs(p0,195.98320000000004,175.1744, 0), v100, z5, tool0;
MoveL Offs(p0,193.975,176.4125, 0), v100, z5, tool0;
MoveL Offs(p0,191.7568,177.4376, 0), v100, z5, tool0;
MoveL Offs(p0,189.3394,178.24429999999998, 0), v100, z5, tool0;
MoveL Offs(p0,186.73360000000002,178.8272, 0), v100, z5, tool0;
MoveL Offs(p0,183.95020000000002,179.1809, 0), v100, z5, tool0;
MoveL Offs(p0,181.0,179.3, 0), v100, z5, tool0;
MoveL Offs(p0,176.71520000000004,179.08640000000003, 0), v100, z5, tool0;
MoveL Offs(p0,174.81879999999995,178.7816, 0), v100, z5, tool0;
MoveL Offs(p0,173.0016,178.3112, 0), v100, z5, tool0;
MoveL Offs(p0,171.2,177.65, 0), v100, z5, tool0;
MoveL Offs(p0,169.35039999999998,176.77280000000002, 0), v100, z5, tool0;
MoveL Offs(p0,167.3892,175.65439999999998, 0), v100, z5, tool0;
MoveL Offs(p0,165.25280000000004,174.26960000000003, 0), v100, z5, tool0;
MoveL Offs(p0,162.8776,172.5932, 0), v100, z5, tool0;
MoveL Offs(p0,160.2,170.6, 0), v100, z5, tool0;
MoveL Offs(p0,157.36830000000003,168.5541, 0), v100, z5, tool0;
MoveL Offs(p0,154.85040000000004,166.97680000000003, 0), v100, z5, tool0;
MoveL Offs(p0,152.6121,165.8687, 0), v100, z5, tool0;
MoveL Offs(p0,150.6192,165.2304, 0), v100, z5, tool0;
MoveL Offs(p0,148.8375,165.0625, 0), v100, z5, tool0;
MoveL Offs(p0,147.2328,165.3656, 0), v100, z5, tool0;
MoveL Offs(p0,145.77089999999998,166.1403, 0), v100, z5, tool0;
MoveL Offs(p0,144.4176,167.3872, 0), v100, z5, tool0;
MoveL Offs(p0,143.1387,169.10690000000002, 0), v100, z5, tool0;
MoveL Offs(p0,141.9,171.3, 0), v100, z5, tool0;
MoveL Offs(p0,139.76719999999997,174.68620000000004, 0), v100, z5, tool0;
MoveL Offs(p0,136.88560000000004,178.12160000000003, 0), v100, z5, tool0;
MoveL Offs(p0,133.4004,181.51139999999998, 0), v100, z5, tool0;
MoveL Offs(p0,129.4568,184.76080000000002, 0), v100, z5, tool0;
MoveL Offs(p0,125.2,187.775, 0), v100, z5, tool0;
MoveL Offs(p0,120.7752,190.4592, 0), v100, z5, tool0;
MoveL Offs(p0,116.32759999999999,192.7186, 0), v100, z5, tool0;
MoveL Offs(p0,112.0024,194.4584, 0), v100, z5, tool0;
MoveL Offs(p0,107.94480000000001,195.58380000000002, 0), v100, z5, tool0;
MoveL Offs(p0,104.3,196.0, 0), v100, z5, tool0;
MoveL Offs(p0,102.46320000000003,196.22320000000005, 0), v100, z5, tool0;
MoveL Offs(p0,102.1598,196.5103, 0), v100, z5, tool0;
MoveL Offs(p0,102.2776,196.9216, 0), v100, z5, tool0;
MoveL Offs(p0,102.825,197.4625, 0), v100, z5, tool0;
MoveL Offs(p0,103.8104,198.1384, 0), v100, z5, tool0;
MoveL Offs(p0,105.2422,198.9547, 0), v100, z5, tool0;
MoveL Offs(p0,107.1288,199.91680000000002, 0), v100, z5, tool0;
MoveL Offs(p0,109.4786,201.0301, 0), v100, z5, tool0;
MoveL Offs(p0,112.3,202.3, 0), v100, z5, tool0;
MoveL Offs(p0,120.35470000000001,205.7833, 0), v100, z5, tool0;
MoveL Offs(p0,128.60560000000004,209.13040000000007, 0), v100, z5, tool0;
MoveL Offs(p0,136.9429,212.3071, 0), v100, z5, tool0;
MoveL Offs(p0,145.25680000000003,215.2792, 0), v100, z5, tool0;
MoveL Offs(p0,153.4375,218.0125, 0), v100, z5, tool0;
MoveL Offs(p0,161.3752,220.4728, 0), v100, z5, tool0;
MoveL Offs(p0,168.9601,222.6259, 0), v100, z5, tool0;
MoveL Offs(p0,176.0824,224.43760000000003, 0), v100, z5, tool0;
MoveL Offs(p0,182.63230000000001,225.8737, 0), v100, z5, tool0;
MoveL Offs(p0,188.5,226.9, 0), v100, z5, tool0;
MoveL Offs(p0,190.811,227.2029, 0), v100, z5, tool0;
MoveL Offs(p0,193.21200000000005,227.45120000000006, 0), v100, z5, tool0;
MoveL Offs(p0,195.655,227.64430000000002, 0), v100, z5, tool0;
MoveL Offs(p0,198.09200000000004,227.78160000000003, 0), v100, z5, tool0;
MoveL Offs(p0,200.475,227.8625, 0), v100, z5, tool0;
MoveL Offs(p0,202.75600000000003,227.8864, 0), v100, z5, tool0;
MoveL Offs(p0,204.887,227.8527, 0), v100, z5, tool0;
MoveL Offs(p0,206.82000000000002,227.76080000000002, 0), v100, z5, tool0;
MoveL Offs(p0,208.507,227.61010000000002, 0), v100, z5, tool0;
MoveL Offs(p0,209.9,227.4, 0), v100, z5, tool0;
MoveL Offs(p0,209.9,227.4, 0), v100, z5, tool0;
MoveJ Offs(p0,27.7,214.9, 10), v100, z1, tool0;
MoveL Offs(p0,27.415600000000005,213.2641, 0), v100, z5, tool0;
MoveL Offs(p0,26.948800000000006,211.36480000000006, 0), v100, z5, tool0;
MoveL Offs(p0,26.339199999999998,209.3047, 0), v100, z5, tool0;
MoveL Offs(p0,25.6264,207.1864, 0), v100, z5, tool0;
MoveL Offs(p0,24.85,205.1125, 0), v100, z5, tool0;
MoveL Offs(p0,24.049599999999995,203.18559999999997, 0), v100, z5, tool0;
MoveL Offs(p0,23.2648,201.50830000000002, 0), v100, z5, tool0;
MoveL Offs(p0,22.535200000000003,200.1832, 0), v100, z5, tool0;
MoveL Offs(p0,21.9004,199.3129, 0), v100, z5, tool0;
MoveL Offs(p0,21.4,199.0, 0), v100, z5, tool0;
MoveL Offs(p0,21.186699999999995,199.5454, 0), v100, z5, tool0;
MoveL Offs(p0,21.142400000000002,199.94080000000002, 0), v100, z5, tool0;
MoveL Offs(p0,21.1125,200.425, 0), v100, z5, tool0;
MoveL Offs(p0,21.0976,200.98719999999997, 0), v100, z5, tool0;
MoveL Offs(p0,21.098300000000002,201.6166, 0), v100, z5, tool0;
MoveL Offs(p0,21.1152,202.30240000000003, 0), v100, z5, tool0;
MoveL Offs(p0,21.148900000000005,203.0338, 0), v100, z5, tool0;
MoveL Offs(p0,21.2,203.8, 0), v100, z5, tool0;
MoveL Offs(p0,21.462900000000005,205.39569999999998, 0), v100, z5, tool0;
MoveL Offs(p0,21.92320000000001,207.28960000000006, 0), v100, z5, tool0;
MoveL Offs(p0,22.5383,209.3719, 0), v100, z5, tool0;
MoveL Offs(p0,23.265600000000003,211.53280000000004, 0), v100, z5, tool0;
MoveL Offs(p0,24.0625,213.6625, 0), v100, z5, tool0;
MoveL Offs(p0,24.8864,215.65119999999996, 0), v100, z5, tool0;
MoveL Offs(p0,25.6947,217.38909999999996, 0), v100, z5, tool0;
MoveL Offs(p0,26.444800000000004,218.76640000000003, 0), v100, z5, tool0;
MoveL Offs(p0,27.094100000000005,219.6733, 0), v100, z5, tool0;
MoveL Offs(p0,27.6,220.0, 0), v100, z5, tool0;
MoveL Offs(p0,27.854699999999998,219.42759999999998, 0), v100, z5, tool0;
MoveL Offs(p0,27.8944,219.0112, 0), v100, z5, tool0;
MoveL Offs(p0,27.9125,218.5, 0), v100, z5, tool0;
MoveL Offs(p0,27.9096,217.90479999999997, 0), v100, z5, tool0;
MoveL Offs(p0,27.8863,217.2364, 0), v100, z5, tool0;
MoveL Offs(p0,27.843200000000003,216.50560000000002, 0), v100, z5, tool0;
MoveL Offs(p0,27.7,214.9, 0), v100, z5, tool0;
MoveJ Offs(p0,250.5,201.8, 10), v100, z1, tool0;
MoveL Offs(p0,250.08150000000006,200.63540000000006, 0), v100, z5, tool0;
MoveL Offs(p0,249.55200000000005,199.43120000000005, 0), v100, z5, tool0;
MoveL Offs(p0,248.92049999999995,198.2018, 0), v100, z5, tool0;
MoveL Offs(p0,248.196,196.96160000000003, 0), v100, z5, tool0;
MoveL Offs(p0,247.3875,195.725, 0), v100, z5, tool0;
MoveL Offs(p0,246.504,194.5064, 0), v100, z5, tool0;
MoveL Offs(p0,245.55450000000002,193.32019999999997, 0), v100, z5, tool0;
MoveL Offs(p0,244.548,192.18080000000003, 0), v100, z5, tool0;
MoveL Offs(p0,243.49349999999998,191.1026, 0), v100, z5, tool0;
MoveL Offs(p0,242.4,190.1, 0), v100, z5, tool0;
MoveL Offs(p0,241.206,189.1107, 0), v100, z5, tool0;
MoveL Offs(p0,239.83200000000005,188.08960000000008, 0), v100, z5, tool0;
MoveL Offs(p0,238.34999999999997,187.07690000000002, 0), v100, z5, tool0;
MoveL Offs(p0,236.83200000000005,186.11280000000005, 0), v100, z5, tool0;
MoveL Offs(p0,235.35,185.2375, 0), v100, z5, tool0;
MoveL Offs(p0,233.97600000000003,184.4912, 0), v100, z5, tool0;
MoveL Offs(p0,232.78199999999998,183.91410000000002, 0), v100, z5, tool0;
MoveL Offs(p0,231.84,183.54640000000003, 0), v100, z5, tool0;
MoveL Offs(p0,231.22200000000004,183.4283, 0), v100, z5, tool0;
MoveL Offs(p0,231.0,183.6, 0), v100, z5, tool0;
MoveL Offs(p0,231.46730000000002,184.8273, 0), v100, z5, tool0;
MoveL Offs(p0,232.74640000000005,186.75840000000005, 0), v100, z5, tool0;
MoveL Offs(p0,234.6531,189.19709999999995, 0), v100, z5, tool0;
MoveL Offs(p0,237.00320000000002,191.9472, 0), v100, z5, tool0;
MoveL Offs(p0,239.6125,194.8125, 0), v100, z5, tool0;
MoveL Offs(p0,242.29680000000002,197.59679999999997, 0), v100, z5, tool0;
MoveL Offs(p0,244.8719,200.10389999999998, 0), v100, z5, tool0;
MoveL Offs(p0,247.1536,202.13760000000002, 0), v100, z5, tool0;
MoveL Offs(p0,248.95770000000002,203.50169999999997, 0), v100, z5, tool0;
MoveL Offs(p0,250.1,204.0, 0), v100, z5, tool0;
MoveL Offs(p0,250.50770000000003,203.7516, 0), v100, z5, tool0;
MoveL Offs(p0,250.5864,203.57120000000003, 0), v100, z5, tool0;
MoveL Offs(p0,250.6375,203.35, 0), v100, z5, tool0;
MoveL Offs(p0,250.6616,203.0928, 0), v100, z5, tool0;
MoveL Offs(p0,250.65929999999997,202.80440000000002, 0), v100, z5, tool0;
MoveL Offs(p0,250.63120000000004,202.48960000000002, 0), v100, z5, tool0;
MoveL Offs(p0,250.5779,202.15320000000003, 0), v100, z5, tool0;
MoveL Offs(p0,250.5,201.8, 0), v100, z5, tool0;
MoveL Offs(p0,250.5,201.8, 0), v100, z5, tool0;
MoveJ Offs(p0,257.5,202.2, 10), v100, z1, tool0;
MoveL Offs(p0,256.1272,202.52960000000002, 0), v100, z5, tool0;
MoveL Offs(p0,255.91240000000002,202.7022, 0), v100, z5, tool0;
MoveL Offs(p0,255.7,202.9, 0), v100, z5, tool0;
MoveL Offs(p0,255.46030000000005,203.1732, 0), v100, z5, tool0;
MoveL Offs(p0,255.2824000000001,203.39360000000005, 0), v100, z5, tool0;
MoveL Offs(p0,255.1681,203.56239999999997, 0), v100, z5, tool0;
MoveL Offs(p0,255.1192,203.6808, 0), v100, z5, tool0;
MoveL Offs(p0,255.1375,203.75, 0), v100, z5, tool0;
MoveL Offs(p0,255.22480000000002,203.7712, 0), v100, z5, tool0;
MoveL Offs(p0,255.3829,203.74560000000002, 0), v100, z5, tool0;
MoveL Offs(p0,255.9187,203.55880000000002, 0), v100, z5, tool0;
MoveL Offs(p0,256.3,203.4, 0), v100, z5, tool0;
MoveL Offs(p0,256.83760000000007,203.18880000000007, 0), v100, z5, tool0;
MoveL Offs(p0,257.0569,203.0652, 0), v100, z5, tool0;
MoveL Offs(p0,257.24080000000004,202.9344, 0), v100, z5, tool0;
MoveL Offs(p0,257.3875,202.8, 0), v100, z5, tool0;
MoveL Offs(p0,257.49519999999995,202.66559999999998, 0), v100, z5, tool0;
MoveL Offs(p0,257.5621,202.5348, 0), v100, z5, tool0;
MoveL Offs(p0,257.5864,202.41120000000004, 0), v100, z5, tool0;
MoveL Offs(p0,257.5663,202.29840000000002, 0), v100, z5, tool0;
MoveL Offs(p0,257.5,202.2, 0), v100, z5, tool0;
MoveL Offs(p0,257.5,202.2, 0), v100, z5, tool0;
MoveJ Offs(p0,262.4,198.8, 10), v100, z1, tool0;
MoveL Offs(p0,262.8021,198.2487, 0), v100, z5, tool0;
MoveL Offs(p0,263.1088000000001,197.78560000000004, 0), v100, z5, tool0;
MoveL Offs(p0,263.32069999999993,197.39690000000002, 0), v100, z5, tool0;
MoveL Offs(p0,263.4384,197.0688, 0), v100, z5, tool0;
MoveL Offs(p0,263.4625,196.7875, 0), v100, z5, tool0;
MoveL Offs(p0,263.3936,196.5392, 0), v100, z5, tool0;
MoveL Offs(p0,263.2323,196.31009999999998, 0), v100, z5, tool0;
MoveL Offs(p0,262.97920000000005,196.0864, 0), v100, z5, tool0;
MoveL Offs(p0,262.6349,195.85430000000002, 0), v100, z5, tool0;
MoveL Offs(p0,262.2,195.6, 0), v100, z5, tool0;
MoveL Offs(p0,261.047,194.83970000000005, 0), v100, z5, tool0;
MoveL Offs(p0,259.8880000000001,193.84960000000004, 0), v100, z5, tool0;
MoveL Offs(p0,258.753,192.6759, 0), v100, z5, tool0;
MoveL Offs(p0,257.672,191.3648, 0), v100, z5, tool0;
MoveL Offs(p0,256.675,189.9625, 0), v100, z5, tool0;
MoveL Offs(p0,255.792,188.5152, 0), v100, z5, tool0;
MoveL Offs(p0,255.05300000000003,187.0691, 0), v100, z5, tool0;
MoveL Offs(p0,254.488,185.67040000000003, 0), v100, z5, tool0;
MoveL Offs(p0,254.12700000000004,184.36530000000002, 0), v100, z5, tool0;
MoveL Offs(p0,254.0,183.2, 0), v100, z5, tool0;
MoveL Offs(p0,253.75,181.7, 0), v100, z5, tool0;
MoveL Offs(p0,253.65439999999998,181.5296, 0), v100, z5, tool0;
MoveL Offs(p0,253.54919999999998,181.41079999999997, 0), v100, z5, tool0;
MoveL Offs(p0,253.43680000000003,181.34720000000002, 0), v100, z5, tool0;
MoveL Offs(p0,253.31959999999998,181.3424, 0), v100, z5, tool0;
MoveL Offs(p0,253.2,181.4, 0), v100, z5, tool0;
MoveL Offs(p0,252.92909999999998,180.84379999999996, 0), v100, z5, tool0;
MoveL Offs(p0,252.88320000000007,180.3296, 0), v100, z5, tool0;
MoveL Offs(p0,252.8625,179.675, 0), v100, z5, tool0;
MoveL Offs(p0,252.86880000000002,178.8944, 0), v100, z5, tool0;
MoveL Offs(p0,252.90389999999996,178.0022, 0), v100, z5, tool0;
MoveL Offs(p0,252.96959999999999,177.01280000000003, 0), v100, z5, tool0;
MoveL Offs(p0,253.52280000000005,172.3059, 0), v100, z5, tool0;
MoveL Offs(p0,254.00640000000007,169.87120000000004, 0), v100, z5, tool0;
MoveL Offs(p0,254.64360000000002,167.50730000000001, 0), v100, z5, tool0;
MoveL Offs(p0,255.4272,165.22560000000001, 0), v100, z5, tool0;
MoveL Offs(p0,256.35,163.0375, 0), v100, z5, tool0;
MoveL Offs(p0,257.40479999999997,160.95440000000002, 0), v100, z5, tool0;
MoveL Offs(p0,258.5844,158.9877, 0), v100, z5, tool0;
MoveL Offs(p0,259.8816,157.14880000000002, 0), v100, z5, tool0;
MoveL Offs(p0,261.28920000000005,155.4491, 0), v100, z5, tool0;
MoveL Offs(p0,262.8,153.9, 0), v100, z5, tool0;
MoveL Offs(p0,263.3751000000001,153.36350000000002, 0), v100, z5, tool0;
MoveL Offs(p0,263.89680000000004,152.89600000000004, 0), v100, z5, tool0;
MoveL Offs(p0,264.3597,152.5005, 0), v100, z5, tool0;
MoveL Offs(p0,264.75840000000005,152.18, 0), v100, z5, tool0;
MoveL Offs(p0,265.0875,151.9375, 0), v100, z5, tool0;
MoveL Offs(p0,265.3416,151.776, 0), v100, z5, tool0;
MoveL Offs(p0,265.5153,151.69850000000002, 0), v100, z5, tool0;
MoveL Offs(p0,265.6032,151.70800000000003, 0), v100, z5, tool0;
MoveL Offs(p0,265.59990000000005,151.8075, 0), v100, z5, tool0;
MoveL Offs(p0,265.5,152.0, 0), v100, z5, tool0;
MoveL Offs(p0,265.8160000000001,152.21200000000005, 0), v100, z5, tool0;
MoveL Offs(p0,266.589,151.757, 0), v100, z5, tool0;
MoveL Offs(p0,267.668,151.008, 0), v100, z5, tool0;
MoveL Offs(p0,268.975,150.025, 0), v100, z5, tool0;
MoveL Offs(p0,270.43199999999996,148.868, 0), v100, z5, tool0;
MoveL Offs(p0,271.96099999999996,147.59699999999998, 0), v100, z5, tool0;
MoveL Offs(p0,273.48400000000004,146.272, 0), v100, z5, tool0;
MoveL Offs(p0,274.923,144.953, 0), v100, z5, tool0;
MoveL Offs(p0,276.2,143.7, 0), v100, z5, tool0;
MoveL Offs(p0,276.66720000000004,143.26870000000002, 0), v100, z5, tool0;
MoveL Offs(p0,277.1056000000001,142.87760000000006, 0), v100, z5, tool0;
MoveL Offs(p0,277.5104,142.5309, 0), v100, z5, tool0;
MoveL Offs(p0,277.8768,142.23280000000003, 0), v100, z5, tool0;
MoveL Offs(p0,278.2,141.9875, 0), v100, z5, tool0;
MoveL Offs(p0,278.4752,141.79919999999998, 0), v100, z5, tool0;
MoveL Offs(p0,278.6976,141.6721, 0), v100, z5, tool0;
MoveL Offs(p0,278.86240000000004,141.6104, 0), v100, z5, tool0;
MoveL Offs(p0,278.9648,141.6183, 0), v100, z5, tool0;
MoveL Offs(p0,279.0,141.7, 0), v100, z5, tool0;
MoveL Offs(p0,280.0336000000001,141.09760000000003, 0), v100, z5, tool0;
MoveL Offs(p0,281.1924,139.9954, 0), v100, z5, tool0;
MoveL Offs(p0,282.6608,138.48880000000003, 0), v100, z5, tool0;
MoveL Offs(p0,284.35,136.675, 0), v100, z5, tool0;
MoveL Offs(p0,286.17119999999994,134.6512, 0), v100, z5, tool0;
MoveL Offs(p0,288.0356,132.5146, 0), v100, z5, tool0;
MoveL Offs(p0,289.8544,130.3624, 0), v100, z5, tool0;
MoveL Offs(p0,291.5388,128.29180000000002, 0), v100, z5, tool0;
MoveL Offs(p0,293.0,126.4, 0), v100, z5, tool0;
MoveL Offs(p0,296.3684,121.51680000000002, 0), v100, z5, tool0;
MoveL Offs(p0,299.3792,116.33840000000005, 0), v100, z5, tool0;
MoveL Offs(p0,302.01079999999996,110.9416, 0), v100, z5, tool0;
MoveL Offs(p0,304.2416,105.40320000000001, 0), v100, z5, tool0;
MoveL Offs(p0,306.05,99.8, 0), v100, z5, tool0;
MoveL Offs(p0,307.4144,94.2088, 0), v100, z5, tool0;
MoveL Offs(p0,308.31319999999994,88.70639999999999, 0), v100, z5, tool0;
MoveL Offs(p0,308.7248000000001,83.36960000000002, 0), v100, z5, tool0;
MoveL Offs(p0,308.6276,78.2752, 0), v100, z5, tool0;
MoveL Offs(p0,308.0,73.5, 0), v100, z5, tool0;
MoveL Offs(p0,307.6320000000001,71.48320000000002, 0), v100, z5, tool0;
MoveL Offs(p0,307.44649999999996,70.47329999999998, 0), v100, z5, tool0;
MoveL Offs(p0,307.264,69.4856, 0), v100, z5, tool0;
MoveL Offs(p0,307.0875,68.5375, 0), v100, z5, tool0;
MoveL Offs(p0,306.91999999999996,67.6464, 0), v100, z5, tool0;
MoveL Offs(p0,306.7645,66.8297, 0), v100, z5, tool0;
MoveL Offs(p0,306.6240000000001,66.1048, 0), v100, z5, tool0;
MoveL Offs(p0,306.5015,65.48910000000001, 0), v100, z5, tool0;
MoveL Offs(p0,306.4,65.0, 0), v100, z5, tool0;
MoveL Offs(p0,306.04910000000007,63.62890000000001, 0), v100, z5, tool0;
MoveL Offs(p0,305.4528000000001,61.92720000000001, 0), v100, z5, tool0;
MoveL Offs(p0,304.6657,60.002300000000005, 0), v100, z5, tool0;
MoveL Offs(p0,303.74240000000003,57.96160000000001, 0), v100, z5, tool0;
MoveL Offs(p0,302.7375,55.9125, 0), v100, z5, tool0;
MoveL Offs(p0,301.7056,53.9624, 0), v100, z5, tool0;
MoveL Offs(p0,300.7013,52.2187, 0), v100, z5, tool0;
MoveL Offs(p0,299.77920000000006,50.7888, 0), v100, z5, tool0;
MoveL Offs(p0,298.99390000000005,49.780100000000004, 0), v100, z5, tool0;
MoveL Offs(p0,298.4,49.3, 0), v100, z5, tool0;
MoveL Offs(p0,297.94720000000007,49.07520000000001, 0), v100, z5, tool0;
MoveL Offs(p0,297.7448,48.9328, 0), v100, z5, tool0;
MoveL Offs(p0,297.5616,48.7736, 0), v100, z5, tool0;
MoveL Offs(p0,297.4,48.6, 0), v100, z5, tool0;
MoveL Offs(p0,297.26239999999996,48.4144, 0), v100, z5, tool0;
MoveL Offs(p0,297.15119999999996,48.2192, 0), v100, z5, tool0;
MoveL Offs(p0,297.0688,48.0168, 0), v100, z5, tool0;
MoveL Offs(p0,297.0176,47.8096, 0), v100, z5, tool0;
MoveL Offs(p0,297.0,47.6, 0), v100, z5, tool0;
MoveL Offs(p0,296.2936000000001,46.39280000000001, 0), v100, z5, tool0;
MoveL Offs(p0,295.49339999999995,45.4967, 0), v100, z5, tool0;
MoveL Offs(p0,294.4688,44.4704, 0), v100, z5, tool0;
MoveL Offs(p0,293.275,43.3625, 0), v100, z5, tool0;
MoveL Offs(p0,291.9672,42.2216, 0), v100, z5, tool0;
MoveL Offs(p0,290.6006,41.0963, 0), v100, z5, tool0;
MoveL Offs(p0,289.23040000000003,40.0352, 0), v100, z5, tool0;
MoveL Offs(p0,287.91179999999997,39.0869, 0), v100, z5, tool0;
MoveL Offs(p0,286.7,38.3, 0), v100, z5, tool0;
MoveL Offs(p0,284.2758,36.98360000000001, 0), v100, z5, tool0;
MoveL Offs(p0,281.87440000000004,35.856800000000014, 0), v100, z5, tool0;
MoveL Offs(p0,279.51259999999996,34.923199999999994, 0), v100, z5, tool0;
MoveL Offs(p0,277.2072,34.186400000000006, 0), v100, z5, tool0;
MoveL Offs(p0,274.975,33.65, 0), v100, z5, tool0;
MoveL Offs(p0,272.8328,33.317600000000006, 0), v100, z5, tool0;
MoveL Offs(p0,270.79740000000004,33.1928, 0), v100, z5, tool0;
MoveL Offs(p0,268.8856,33.2792, 0), v100, z5, tool0;
MoveL Offs(p0,267.11420000000004,33.580400000000004, 0), v100, z5, tool0;
MoveL Offs(p0,265.5,34.1, 0), v100, z5, tool0;
MoveL Offs(p0,265.0213,34.3066, 0), v100, z5, tool0;
MoveL Offs(p0,264.5504000000001,34.5048, 0), v100, z5, tool0;
MoveL Offs(p0,264.09510000000006,34.69219999999999, 0), v100, z5, tool0;
MoveL Offs(p0,263.6632,34.866400000000006, 0), v100, z5, tool0;
MoveL Offs(p0,263.2625,35.025, 0), v100, z5, tool0;
MoveL Offs(p0,262.9008,35.1656, 0), v100, z5, tool0;
MoveL Offs(p0,262.5859,35.2858, 0), v100, z5, tool0;
MoveL Offs(p0,262.3256,35.3832, 0), v100, z5, tool0;
MoveL Offs(p0,262.1277,35.4554, 0), v100, z5, tool0;
MoveL Offs(p0,262.0,35.5, 0), v100, z5, tool0;
MoveL Offs(p0,261.28370000000007,35.769800000000004, 0), v100, z5, tool0;
MoveL Offs(p0,260.6376000000001,36.03840000000001, 0), v100, z5, tool0;
MoveL Offs(p0,260.0659,36.3046, 0), v100, z5, tool0;
MoveL Offs(p0,259.57280000000003,36.5672, 0), v100, z5, tool0;
MoveL Offs(p0,259.1625,36.825, 0), v100, z5, tool0;
MoveL Offs(p0,258.8392,37.0768, 0), v100, z5, tool0;
MoveL Offs(p0,258.6071,37.3214, 0), v100, z5, tool0;
MoveL Offs(p0,258.47040000000004,37.5576, 0), v100, z5, tool0;
MoveL Offs(p0,258.43330000000003,37.7842, 0), v100, z5, tool0;
MoveL Offs(p0,258.5,38.0, 0), v100, z5, tool0;
MoveL Offs(p0,258.1598,38.9625, 0), v100, z5, tool0;
MoveL Offs(p0,257.99120000000005,39.088, 0), v100, z5, tool0;
MoveL Offs(p0,257.8034,39.201499999999996, 0), v100, z5, tool0;
MoveL Offs(p0,257.6,39.3, 0), v100, z5, tool0;
MoveL Offs(p0,257.0792,39.592000000000006, 0), v100, z5, tool0;
MoveL Offs(p0,256.7963,39.813, 0), v100, z5, tool0;
MoveL Offs(p0,256.5056,40.07600000000001, 0), v100, z5, tool0;
MoveL Offs(p0,256.2125,40.375, 0), v100, z5, tool0;
MoveL Offs(p0,255.9224,40.70399999999999, 0), v100, z5, tool0;
MoveL Offs(p0,255.6407,41.057, 0), v100, z5, tool0;
MoveL Offs(p0,255.3728,41.42800000000001, 0), v100, z5, tool0;
MoveL Offs(p0,255.1241,41.811, 0), v100, z5, tool0;
MoveL Offs(p0,254.9,42.2, 0), v100, z5, tool0;
MoveL Offs(p0,254.67000000000002,42.67960000000001, 0), v100, z5, tool0;
MoveL Offs(p0,254.52400000000011,43.036800000000014, 0), v100, z5, tool0;
MoveL Offs(p0,254.468,43.2692, 0), v100, z5, tool0;
MoveL Offs(p0,254.50799999999998,43.374399999999994, 0), v100, z5, tool0;
MoveL Offs(p0,254.65,43.35, 0), v100, z5, tool0;
MoveL Offs(p0,255.26399999999998,42.9028, 0), v100, z5, tool0;
MoveL Offs(p0,255.74800000000005,42.47520000000001, 0), v100, z5, tool0;
MoveL Offs(p0,256.358,41.9084, 0), v100, z5, tool0;
MoveL Offs(p0,257.1,41.2, 0), v100, z5, tool0;
MoveL Offs(p0,258.58250000000004,39.8206, 0), v100, z5, tool0;
MoveL Offs(p0,259.9360000000001,38.67280000000001, 0), v100, z5, tool0;
MoveL Offs(p0,261.1995,37.7422, 0), v100, z5, tool0;
MoveL Offs(p0,262.41200000000003,37.0144, 0), v100, z5, tool0;
MoveL Offs(p0,263.6125,36.475, 0), v100, z5, tool0;
MoveL Offs(p0,264.84000000000003,36.10960000000001, 0), v100, z5, tool0;
MoveL Offs(p0,266.1335,35.903800000000004, 0), v100, z5, tool0;
MoveL Offs(p0,267.53200000000004,35.8432, 0), v100, z5, tool0;
MoveL Offs(p0,269.0745,35.9134, 0), v100, z5, tool0;
MoveL Offs(p0,270.8,36.1, 0), v100, z5, tool0;
MoveL Offs(p0,273.0074,36.494200000000006, 0), v100, z5, tool0;
MoveL Offs(p0,275.2352,37.069600000000015, 0), v100, z5, tool0;
MoveL Offs(p0,277.4618,37.8154, 0), v100, z5, tool0;
MoveL Offs(p0,279.6656,38.720800000000004, 0), v100, z5, tool0;
MoveL Offs(p0,281.825,39.775, 0), v100, z5, tool0;
MoveL Offs(p0,283.91839999999996,40.9672, 0), v100, z5, tool0;
MoveL Offs(p0,285.92420000000004,42.2866, 0), v100, z5, tool0;
MoveL Offs(p0,287.8208000000001,43.72240000000001, 0), v100, z5, tool0;
MoveL Offs(p0,289.58660000000003,45.2638, 0), v100, z5, tool0;
MoveL Offs(p0,291.2,46.9, 0), v100, z5, tool0;
MoveL Offs(p0,292.53990000000005,48.42920000000001, 0), v100, z5, tool0;
MoveL Offs(p0,293.8432000000001,50.04960000000001, 0), v100, z5, tool0;
MoveL Offs(p0,295.0853,51.7204, 0), v100, z5, tool0;
MoveL Offs(p0,296.2416,53.40080000000002, 0), v100, z5, tool0;
MoveL Offs(p0,297.2875,55.05, 0), v100, z5, tool0;
MoveL Offs(p0,298.1984,56.6272, 0), v100, z5, tool0;
MoveL Offs(p0,298.9497,58.09160000000001, 0), v100, z5, tool0;
MoveL Offs(p0,299.51680000000005,59.402400000000014, 0), v100, z5, tool0;
MoveL Offs(p0,299.87510000000003,60.5188, 0), v100, z5, tool0;
MoveL Offs(p0,300.0,61.4, 0), v100, z5, tool0;
MoveL Offs(p0,300.256,62.529599999999995, 0), v100, z5, tool0;
MoveL Offs(p0,300.3875,62.8375, 0), v100, z5, tool0;
MoveL Offs(p0,300.54,63.142399999999995, 0), v100, z5, tool0;
MoveL Offs(p0,300.7105,63.43769999999999, 0), v100, z5, tool0;
MoveL Offs(p0,300.8960000000001,63.7168, 0), v100, z5, tool0;
MoveL Offs(p0,301.09350000000006,63.9731, 0), v100, z5, tool0;
MoveL Offs(p0,301.3,64.2, 0), v100, z5, tool0;
MoveL Offs(p0,301.7151,64.7077, 0), v100, z5, tool0;
MoveL Offs(p0,302.0648000000001,65.30960000000002, 0), v100, z5, tool0;
MoveL Offs(p0,302.35569999999996,66.06389999999999, 0), v100, z5, tool0;
MoveL Offs(p0,302.59440000000006,67.0288, 0), v100, z5, tool0;
MoveL Offs(p0,302.7875,68.2625, 0), v100, z5, tool0;
MoveL Offs(p0,302.9416,69.8232, 0), v100, z5, tool0;
MoveL Offs(p0,303.06329999999997,71.76910000000001, 0), v100, z5, tool0;
MoveL Offs(p0,303.15920000000006,74.1584, 0), v100, z5, tool0;
MoveL Offs(p0,303.2359,77.04929999999999, 0), v100, z5, tool0;
MoveL Offs(p0,303.3,80.5, 0), v100, z5, tool0;
MoveL Offs(p0,303.0792,87.468, 0), v100, z5, tool0;
MoveL Offs(p0,302.9625,89.1875, 0), v100, z5, tool0;
MoveL Offs(p0,302.8248,90.832, 0), v100, z5, tool0;
MoveL Offs(p0,302.66790000000003,92.36850000000001, 0), v100, z5, tool0;
MoveL Offs(p0,302.4936,93.76400000000001, 0), v100, z5, tool0;
MoveL Offs(p0,302.30370000000005,94.98550000000002, 0), v100, z5, tool0;
MoveL Offs(p0,302.1,96.0, 0), v100, z5, tool0;
MoveL Offs(p0,301.5896,97.8452, 0), v100, z5, tool0;
MoveL Offs(p0,300.8728000000001,100.05760000000002, 0), v100, z5, tool0;
MoveL Offs(p0,300.0012,102.5124, 0), v100, z5, tool0;
MoveL Offs(p0,299.0264,105.08480000000002, 0), v100, z5, tool0;
MoveL Offs(p0,298.0,107.65, 0), v100, z5, tool0;
MoveL Offs(p0,296.9736,110.0832, 0), v100, z5, tool0;
MoveL Offs(p0,295.9988,112.2596, 0), v100, z5, tool0;
MoveL Offs(p0,295.1272,114.05440000000003, 0), v100, z5, tool0;
MoveL Offs(p0,294.41040000000004,115.34280000000001, 0), v100, z5, tool0;
MoveL Offs(p0,293.9,116.0, 0), v100, z5, tool0;
MoveL Offs(p0,293.6544000000001,116.29280000000003, 0), v100, z5, tool0;
MoveL Offs(p0,293.4896,116.51570000000001, 0), v100, z5, tool0;
MoveL Offs(p0,293.3032,116.78240000000001, 0), v100, z5, tool0;
MoveL Offs(p0,293.1,117.0875, 0), v100, z5, tool0;
MoveL Offs(p0,292.8848,117.4256, 0), v100, z5, tool0;
MoveL Offs(p0,292.66240000000005,117.7913, 0), v100, z5, tool0;
MoveL Offs(p0,292.43760000000003,118.17920000000001, 0), v100, z5, tool0;
MoveL Offs(p0,292.2152,118.5839, 0), v100, z5, tool0;
MoveL Offs(p0,292.0,119.0, 0), v100, z5, tool0;
MoveL Offs(p0,291.73220000000003,119.4804, 0), v100, z5, tool0;
MoveL Offs(p0,291.35760000000005,120.07120000000005, 0), v100, z5, tool0;
MoveL Offs(p0,290.88939999999997,120.7568, 0), v100, z5, tool0;
MoveL Offs(p0,290.34080000000006,121.5216, 0), v100, z5, tool0;
MoveL Offs(p0,289.725,122.35, 0), v100, z5, tool0;
MoveL Offs(p0,289.05519999999996,123.22640000000001, 0), v100, z5, tool0;
MoveL Offs(p0,288.3446,124.13519999999998, 0), v100, z5, tool0;
MoveL Offs(p0,287.6064,125.06080000000001, 0), v100, z5, tool0;
MoveL Offs(p0,286.8538,125.9876, 0), v100, z5, tool0;
MoveL Offs(p0,286.1,126.9, 0), v100, z5, tool0;
MoveL Offs(p0,285.3667000000001,127.7648, 0), v100, z5, tool0;
MoveL Offs(p0,284.6736000000001,128.61040000000003, 0), v100, z5, tool0;
MoveL Offs(p0,284.03090000000003,129.42360000000002, 0), v100, z5, tool0;
MoveL Offs(p0,283.4488,130.1912, 0), v100, z5, tool0;
MoveL Offs(p0,282.9375,130.9, 0), v100, z5, tool0;
MoveL Offs(p0,282.5072,131.5368, 0), v100, z5, tool0;
MoveL Offs(p0,282.1681,132.0884, 0), v100, z5, tool0;
MoveL Offs(p0,281.9304,132.54160000000002, 0), v100, z5, tool0;
MoveL Offs(p0,281.8043,132.88320000000002, 0), v100, z5, tool0;
MoveL Offs(p0,281.8,133.1, 0), v100, z5, tool0;
MoveL Offs(p0,281.59119999999996,133.74079999999998, 0), v100, z5, tool0;
MoveL Offs(p0,281.4906,133.7874, 0), v100, z5, tool0;
MoveL Offs(p0,281.37440000000004,133.8136, 0), v100, z5, tool0;
MoveL Offs(p0,281.2438,133.8182, 0), v100, z5, tool0;
MoveL Offs(p0,281.1,133.8, 0), v100, z5, tool0;
MoveL Offs(p0,279.9858,134.26799999999997, 0), v100, z5, tool0;
MoveL Offs(p0,279.3576,134.68, 0), v100, z5, tool0;
MoveL Offs(p0,278.625,135.2, 0), v100, z5, tool0;
MoveL Offs(p0,277.8024,135.81599999999997, 0), v100, z5, tool0;
MoveL Offs(p0,276.9042,136.516, 0), v100, z5, tool0;
MoveL Offs(p0,275.94480000000004,137.288, 0), v100, z5, tool0;
MoveL Offs(p0,274.9386,138.12, 0), v100, z5, tool0;
MoveL Offs(p0,273.9,139.0, 0), v100, z5, tool0;
MoveL Offs(p0,272.83220000000006,139.93350000000004, 0), v100, z5, tool0;
MoveL Offs(p0,271.74160000000006,140.86400000000006, 0), v100, z5, tool0;
MoveL Offs(p0,270.64739999999995,141.7765, 0), v100, z5, tool0;
MoveL Offs(p0,269.5688,142.656, 0), v100, z5, tool0;
MoveL Offs(p0,268.525,143.4875, 0), v100, z5, tool0;
MoveL Offs(p0,267.5352,144.256, 0), v100, z5, tool0;
MoveL Offs(p0,266.61859999999996,144.9465, 0), v100, z5, tool0;
MoveL Offs(p0,265.7944,145.544, 0), v100, z5, tool0;
MoveL Offs(p0,265.08180000000004,146.0335, 0), v100, z5, tool0;
MoveL Offs(p0,264.5,146.4, 0), v100, z5, tool0;
MoveL Offs(p0,263.10880000000003,147.3563, 0), v100, z5, tool0;
MoveL Offs(p0,261.61440000000005,148.50640000000004, 0), v100, z5, tool0;
MoveL Offs(p0,260.0756,149.79209999999998, 0), v100, z5, tool0;
MoveL Offs(p0,258.5512,151.1552, 0), v100, z5, tool0;
MoveL Offs(p0,257.1,152.5375, 0), v100, z5, tool0;
MoveL Offs(p0,255.7808,153.8808, 0), v100, z5, tool0;
MoveL Offs(p0,254.6524,155.1269, 0), v100, z5, tool0;
MoveL Offs(p0,253.7736,156.2176, 0), v100, z5, tool0;
MoveL Offs(p0,253.2032,157.09470000000002, 0), v100, z5, tool0;
MoveL Offs(p0,253.0,157.7, 0), v100, z5, tool0;
MoveL Offs(p0,252.75,158.6125, 0), v100, z5, tool0;
MoveL Offs(p0,252.65439999999998,158.744, 0), v100, z5, tool0;
MoveL Offs(p0,252.54919999999998,158.85150000000002, 0), v100, z5, tool0;
MoveL Offs(p0,252.43680000000003,158.93200000000002, 0), v100, z5, tool0;
MoveL Offs(p0,252.31959999999998,158.98250000000002, 0), v100, z5, tool0;
MoveL Offs(p0,252.2,159.0, 0), v100, z5, tool0;
MoveL Offs(p0,251.66930000000002,159.2982, 0), v100, z5, tool0;
MoveL Offs(p0,251.11040000000008,160.13760000000005, 0), v100, z5, tool0;
MoveL Offs(p0,250.5431,161.43540000000002, 0), v100, z5, tool0;
MoveL Offs(p0,249.98720000000003,163.10880000000003, 0), v100, z5, tool0;
MoveL Offs(p0,249.4625,165.075, 0), v100, z5, tool0;
MoveL Offs(p0,248.9888,167.25119999999998, 0), v100, z5, tool0;
MoveL Offs(p0,248.58589999999998,169.5546, 0), v100, z5, tool0;
MoveL Offs(p0,248.2736,171.9024, 0), v100, z5, tool0;
MoveL Offs(p0,248.07170000000002,174.21179999999998, 0), v100, z5, tool0;
MoveL Offs(p0,248.0,176.4, 0), v100, z5, tool0;
MoveL Offs(p0,248.25680000000003,181.52720000000005, 0), v100, z5, tool0;
MoveL Offs(p0,248.58319999999998,183.8583, 0), v100, z5, tool0;
MoveL Offs(p0,249.0464,186.0496, 0), v100, z5, tool0;
MoveL Offs(p0,249.65,188.1125, 0), v100, z5, tool0;
MoveL Offs(p0,250.3976,190.05839999999998, 0), v100, z5, tool0;
MoveL Offs(p0,251.2928,191.89870000000002, 0), v100, z5, tool0;
MoveL Offs(p0,252.33920000000003,193.64480000000003, 0), v100, z5, tool0;
MoveL Offs(p0,253.5404,195.30810000000002, 0), v100, z5, tool0;
MoveL Offs(p0,254.9,196.9, 0), v100, z5, tool0;
MoveL Offs(p0,256.0982,198.17900000000003, 0), v100, z5, tool0;
MoveL Offs(p0,257.1296000000001,199.20000000000005, 0), v100, z5, tool0;
MoveL Offs(p0,258.0194,199.969, 0), v100, z5, tool0;
MoveL Offs(p0,258.79280000000006,200.49200000000002, 0), v100, z5, tool0;
MoveL Offs(p0,259.475,200.775, 0), v100, z5, tool0;
MoveL Offs(p0,260.0912,200.824, 0), v100, z5, tool0;
MoveL Offs(p0,260.6666,200.64499999999998, 0), v100, z5, tool0;
MoveL Offs(p0,261.2264,200.244, 0), v100, z5, tool0;
MoveL Offs(p0,261.7958,199.627, 0), v100, z5, tool0;
MoveL Offs(p0,262.4,198.8, 0), v100, z5, tool0;
MoveL Offs(p0,262.4,198.8, 0), v100, z5, tool0;
MoveJ Offs(p0,36.2,197.9, 10), v100, z1, tool0;
MoveL Offs(p0,37.53840000000001,197.48960000000005, 0), v100, z5, tool0;
MoveL Offs(p0,38.246599999999994,197.21239999999995, 0), v100, z5, tool0;
MoveL Offs(p0,38.96320000000001,196.8968, 0), v100, z5, tool0;
MoveL Offs(p0,39.675,196.55, 0), v100, z5, tool0;
MoveL Offs(p0,40.3688,196.17919999999998, 0), v100, z5, tool0;
MoveL Offs(p0,41.0314,195.79159999999996, 0), v100, z5, tool0;
MoveL Offs(p0,41.64960000000001,195.3944, 0), v100, z5, tool0;
MoveL Offs(p0,42.2102,194.9948, 0), v100, z5, tool0;
MoveL Offs(p0,42.7,194.6, 0), v100, z5, tool0;
MoveL Offs(p0,45.4,192.2, 0), v100, z5, tool0;
MoveL Offs(p0,41.7,188.1, 0), v100, z5, tool0;
MoveL Offs(p0,41.036500000000004,187.32710000000003, 0), v100, z5, tool0;
MoveL Offs(p0,40.31600000000002,186.40480000000002, 0), v100, z5, tool0;
MoveL Offs(p0,39.5535,185.3577, 0), v100, z5, tool0;
MoveL Offs(p0,38.763999999999996,184.2104, 0), v100, z5, tool0;
MoveL Offs(p0,37.9625,182.9875, 0), v100, z5, tool0;
MoveL Offs(p0,37.164,181.71359999999999, 0), v100, z5, tool0;
MoveL Offs(p0,36.3835,180.41330000000002, 0), v100, z5, tool0;
MoveL Offs(p0,35.636,179.1112, 0), v100, z5, tool0;
MoveL Offs(p0,34.9365,177.83190000000002, 0), v100, z5, tool0;
MoveL Offs(p0,34.3,176.6, 0), v100, z5, tool0;
MoveL Offs(p0,33.3198,174.5941, 0), v100, z5, tool0;
MoveL Offs(p0,32.50640000000001,172.98480000000006, 0), v100, z5, tool0;
MoveL Offs(p0,31.8106,171.72469999999998, 0), v100, z5, tool0;
MoveL Offs(p0,31.183200000000006,170.76640000000003, 0), v100, z5, tool0;
MoveL Offs(p0,30.575,170.0625, 0), v100, z5, tool0;
MoveL Offs(p0,29.936799999999998,169.5656, 0), v100, z5, tool0;
MoveL Offs(p0,29.219399999999997,169.2283, 0), v100, z5, tool0;
MoveL Offs(p0,28.3736,169.00320000000002, 0), v100, z5, tool0;
MoveL Offs(p0,27.3502,168.84290000000001, 0), v100, z5, tool0;
MoveL Offs(p0,26.1,168.7, 0), v100, z5, tool0;
MoveL Offs(p0,23.8284,168.4309, 0), v100, z5, tool0;
MoveL Offs(p0,23.0968,168.3128, 0), v100, z5, tool0;
MoveL Offs(p0,22.4,168.1875, 0), v100, z5, tool0;
MoveL Offs(p0,21.7512,168.0592, 0), v100, z5, tool0;
MoveL Offs(p0,21.163599999999995,167.9321, 0), v100, z5, tool0;
MoveL Offs(p0,20.6504,167.81040000000002, 0), v100, z5, tool0;
MoveL Offs(p0,20.224800000000002,167.6983, 0), v100, z5, tool0;
MoveL Offs(p0,19.9,167.6, 0), v100, z5, tool0;
MoveL Offs(p0,18.901899999999998,167.81329999999997, 0), v100, z5, tool0;
MoveL Offs(p0,18.664800000000003,168.34560000000005, 0), v100, z5, tool0;
MoveL Offs(p0,18.4625,169.1875, 0), v100, z5, tool0;
MoveL Offs(p0,18.287200000000002,170.3864, 0), v100, z5, tool0;
MoveL Offs(p0,18.131099999999996,171.9897, 0), v100, z5, tool0;
MoveL Offs(p0,17.986400000000003,174.04480000000004, 0), v100, z5, tool0;
MoveL Offs(p0,17.8453,176.5991, 0), v100, z5, tool0;
MoveL Offs(p0,17.7,179.7, 0), v100, z5, tool0;
MoveL Offs(p0,17.2,192.5, 0), v100, z5, tool0;
MoveL Offs(p0,19.8,194.8, 0), v100, z5, tool0;
MoveL Offs(p0,21.260900000000003,195.9857, 0), v100, z5, tool0;
MoveL Offs(p0,22.715200000000003,196.96560000000005, 0), v100, z5, tool0;
MoveL Offs(p0,24.180300000000003,197.7439, 0), v100, z5, tool0;
MoveL Offs(p0,25.6736,198.3248, 0), v100, z5, tool0;
MoveL Offs(p0,27.2125,198.7125, 0), v100, z5, tool0;
MoveL Offs(p0,28.8144,198.91119999999998, 0), v100, z5, tool0;
MoveL Offs(p0,30.496699999999997,198.9251, 0), v100, z5, tool0;
MoveL Offs(p0,32.2768,198.75840000000002, 0), v100, z5, tool0;
MoveL Offs(p0,34.1721,198.41530000000003, 0), v100, z5, tool0;
MoveL Offs(p0,36.2,197.9, 0), v100, z5, tool0;
MoveL Offs(p0,36.2,197.9, 0), v100, z5, tool0;
MoveJ Offs(p0,15.8,177.2, 10), v100, z1, tool0;
MoveL Offs(p0,15.5,165.4, 0), v100, z5, tool0;
MoveL Offs(p0,12.0,162.3, 0), v100, z5, tool0;
MoveL Offs(p0,11.434500000000003,161.8032, 0), v100, z5, tool0;
MoveL Offs(p0,10.884000000000002,161.33760000000004, 0), v100, z5, tool0;
MoveL Offs(p0,10.357499999999998,160.9104, 0), v100, z5, tool0;
MoveL Offs(p0,9.863999999999999,160.5288, 0), v100, z5, tool0;
MoveL Offs(p0,9.4125,160.2, 0), v100, z5, tool0;
MoveL Offs(p0,9.012,159.9312, 0), v100, z5, tool0;
MoveL Offs(p0,8.6715,159.7296, 0), v100, z5, tool0;
MoveL Offs(p0,8.4,159.6024, 0), v100, z5, tool0;
MoveL Offs(p0,8.2065,159.5568, 0), v100, z5, tool0;
MoveL Offs(p0,8.1,159.6, 0), v100, z5, tool0;
MoveL Offs(p0,7.876800000000001,160.17370000000003, 0), v100, z5, tool0;
MoveL Offs(p0,7.742400000000002,161.3336, 0), v100, z5, tool0;
MoveL Offs(p0,7.6896,162.9579, 0), v100, z5, tool0;
MoveL Offs(p0,7.711200000000001,164.9248, 0), v100, z5, tool0;
MoveL Offs(p0,7.8,167.1125, 0), v100, z5, tool0;
MoveL Offs(p0,8.3976,173.7824, 0), v100, z5, tool0;
MoveL Offs(p0,8.683200000000001,175.6353, 0), v100, z5, tool0;
MoveL Offs(p0,9.0,177.1, 0), v100, z5, tool0;
MoveL Offs(p0,9.4975,178.81830000000005, 0), v100, z5, tool0;
MoveL Offs(p0,10.076000000000004,180.52640000000002, 0), v100, z5, tool0;
MoveL Offs(p0,10.7145,182.1841, 0), v100, z5, tool0;
MoveL Offs(p0,11.392000000000001,183.7512, 0), v100, z5, tool0;
MoveL Offs(p0,12.0875,185.1875, 0), v100, z5, tool0;
MoveL Offs(p0,12.78,186.4528, 0), v100, z5, tool0;
MoveL Offs(p0,13.448500000000001,187.5069, 0), v100, z5, tool0;
MoveL Offs(p0,14.072000000000003,188.3096, 0), v100, z5, tool0;
MoveL Offs(p0,14.629500000000002,188.82070000000002, 0), v100, z5, tool0;
MoveL Offs(p0,15.1,189.0, 0), v100, z5, tool0;
MoveL Offs(p0,15.470400000000007,188.53120000000007, 0), v100, z5, tool0;
MoveL Offs(p0,15.616599999999996,187.94429999999997, 0), v100, z5, tool0;
MoveL Offs(p0,15.7352,187.1216, 0), v100, z5, tool0;
MoveL Offs(p0,15.825,186.0625, 0), v100, z5, tool0;
MoveL Offs(p0,15.884799999999998,184.7664, 0), v100, z5, tool0;
MoveL Offs(p0,15.913400000000001,183.23270000000002, 0), v100, z5, tool0;
MoveL Offs(p0,15.909600000000001,181.4608, 0), v100, z5, tool0;
MoveL Offs(p0,15.872200000000001,179.45010000000002, 0), v100, z5, tool0;
MoveL Offs(p0,15.8,177.2, 0), v100, z5, tool0;
MoveL Offs(p0,15.8,177.2, 0), v100, z5, tool0;
MoveJ Offs(p0,47.0,186.6, 10), v100, z1, tool0;
MoveL Offs(p0,46.68400000000001,183.89840000000007, 0), v100, z5, tool0;
MoveL Offs(p0,46.298,182.39159999999998, 0), v100, z5, tool0;
MoveL Offs(p0,45.768,180.80320000000003, 0), v100, z5, tool0;
MoveL Offs(p0,45.1,179.15, 0), v100, z5, tool0;
MoveL Offs(p0,44.3,177.4488, 0), v100, z5, tool0;
MoveL Offs(p0,43.373999999999995,175.71639999999996, 0), v100, z5, tool0;
MoveL Offs(p0,42.327999999999996,173.96960000000004, 0), v100, z5, tool0;
MoveL Offs(p0,41.168,172.2252, 0), v100, z5, tool0;
MoveL Offs(p0,39.9,170.5, 0), v100, z5, tool0;
MoveL Offs(p0,39.2323,169.58120000000002, 0), v100, z5, tool0;
MoveL Offs(p0,38.6144,168.69360000000003, 0), v100, z5, tool0;
MoveL Offs(p0,38.054100000000005,167.8504, 0), v100, z5, tool0;
MoveL Offs(p0,37.5592,167.06480000000002, 0), v100, z5, tool0;
MoveL Offs(p0,37.1375,166.35, 0), v100, z5, tool0;
MoveL Offs(p0,36.7968,165.71919999999997, 0), v100, z5, tool0;
MoveL Offs(p0,36.5449,165.18559999999997, 0), v100, z5, tool0;
MoveL Offs(p0,36.38960000000001,164.7624, 0), v100, z5, tool0;
MoveL Offs(p0,36.3387,164.4628, 0), v100, z5, tool0;
MoveL Offs(p0,36.4,164.3, 0), v100, z5, tool0;
MoveL Offs(p0,37.325,164.5125, 0), v100, z5, tool0;
MoveL Offs(p0,37.588,164.7248, 0), v100, z5, tool0;
MoveL Offs(p0,37.863,164.9839, 0), v100, z5, tool0;
MoveL Offs(p0,38.144000000000005,165.28560000000002, 0), v100, z5, tool0;
MoveL Offs(p0,38.425,165.6257, 0), v100, z5, tool0;
MoveL Offs(p0,38.7,166.0, 0), v100, z5, tool0;
MoveL Offs(p0,39.7128,167.4178, 0), v100, z5, tool0;
MoveL Offs(p0,40.75440000000001,168.77440000000004, 0), v100, z5, tool0;
MoveL Offs(p0,41.7996,170.04459999999997, 0), v100, z5, tool0;
MoveL Offs(p0,42.82320000000001,171.2032, 0), v100, z5, tool0;
MoveL Offs(p0,43.8,172.225, 0), v100, z5, tool0;
MoveL Offs(p0,44.7048,173.0848, 0), v100, z5, tool0;
MoveL Offs(p0,45.5124,173.75740000000002, 0), v100, z5, tool0;
MoveL Offs(p0,46.19760000000001,174.2176, 0), v100, z5, tool0;
MoveL Offs(p0,46.735200000000006,174.4402, 0), v100, z5, tool0;
MoveL Offs(p0,47.1,174.4, 0), v100, z5, tool0;
MoveL Offs(p0,47.512600000000006,174.05070000000003, 0), v100, z5, tool0;
MoveL Offs(p0,47.78480000000001,173.58560000000006, 0), v100, z5, tool0;
MoveL Offs(p0,47.908199999999994,172.9789, 0), v100, z5, tool0;
MoveL Offs(p0,47.8744,172.2048, 0), v100, z5, tool0;
MoveL Offs(p0,47.675,171.2375, 0), v100, z5, tool0;
MoveL Offs(p0,47.30159999999999,170.0512, 0), v100, z5, tool0;
MoveL Offs(p0,46.745799999999996,168.6201, 0), v100, z5, tool0;
MoveL Offs(p0,45.99920000000001,166.91840000000002, 0), v100, z5, tool0;
MoveL Offs(p0,45.0534,164.9203, 0), v100, z5, tool0;
MoveL Offs(p0,43.9,162.6, 0), v100, z5, tool0;
MoveL Offs(p0,43.077600000000004,160.9916, 0), v100, z5, tool0;
MoveL Offs(p0,42.28880000000001,159.52480000000006, 0), v100, z5, tool0;
MoveL Offs(p0,41.5312,158.19719999999998, 0), v100, z5, tool0;
MoveL Offs(p0,40.8024,157.0064, 0), v100, z5, tool0;
MoveL Offs(p0,40.1,155.95, 0), v100, z5, tool0;
MoveL Offs(p0,39.4216,155.0256, 0), v100, z5, tool0;
MoveL Offs(p0,38.7648,154.2308, 0), v100, z5, tool0;
MoveL Offs(p0,38.1272,153.5632, 0), v100, z5, tool0;
MoveL Offs(p0,37.5064,153.02040000000002, 0), v100, z5, tool0;
MoveL Offs(p0,36.9,152.6, 0), v100, z5, tool0;
MoveL Offs(p0,35.74100000000001,151.87830000000002, 0), v100, z5, tool0;
MoveL Offs(p0,34.948000000000015,151.27840000000003, 0), v100, z5, tool0;
MoveL Offs(p0,34.497,150.8081, 0), v100, z5, tool0;
MoveL Offs(p0,34.364000000000004,150.4752, 0), v100, z5, tool0;
MoveL Offs(p0,34.525,150.2875, 0), v100, z5, tool0;
MoveL Offs(p0,34.956,150.2528, 0), v100, z5, tool0;
MoveL Offs(p0,35.632999999999996,150.3789, 0), v100, z5, tool0;
MoveL Offs(p0,36.532000000000004,150.67360000000002, 0), v100, z5, tool0;
MoveL Offs(p0,37.629,151.1447, 0), v100, z5, tool0;
MoveL Offs(p0,38.9,151.8, 0), v100, z5, tool0;
MoveL Offs(p0,39.814400000000006,152.31640000000002, 0), v100, z5, tool0;
MoveL Offs(p0,40.58720000000001,152.72720000000007, 0), v100, z5, tool0;
MoveL Offs(p0,41.232800000000005,153.0348, 0), v100, z5, tool0;
MoveL Offs(p0,41.765600000000006,153.2416, 0), v100, z5, tool0;
MoveL Offs(p0,42.2,153.35, 0), v100, z5, tool0;
MoveL Offs(p0,42.5504,153.36239999999998, 0), v100, z5, tool0;
MoveL Offs(p0,42.831199999999995,153.28119999999998, 0), v100, z5, tool0;
MoveL Offs(p0,43.056799999999996,153.10880000000003, 0), v100, z5, tool0;
MoveL Offs(p0,43.2416,152.8476, 0), v100, z5, tool0;
MoveL Offs(p0,43.4,152.5, 0), v100, z5, tool0;
MoveL Offs(p0,43.18960000000001,149.31600000000003, 0), v100, z5, tool0;
MoveL Offs(p0,42.392900000000004,147.289, 0), v100, z5, tool0;
MoveL Offs(p0,41.2608,145.14800000000002, 0), v100, z5, tool0;
MoveL Offs(p0,39.8875,143.025, 0), v100, z5, tool0;
MoveL Offs(p0,38.367200000000004,141.052, 0), v100, z5, tool0;
MoveL Offs(p0,36.7941,139.361, 0), v100, z5, tool0;
MoveL Offs(p0,35.2624,138.084, 0), v100, z5, tool0;
MoveL Offs(p0,33.8663,137.353, 0), v100, z5, tool0;
MoveL Offs(p0,32.7,137.3, 0), v100, z5, tool0;
MoveL Offs(p0,32.032300000000006,137.7023, 0), v100, z5, tool0;
MoveL Offs(p0,31.41440000000001,138.46640000000002, 0), v100, z5, tool0;
MoveL Offs(p0,30.8541,139.5581, 0), v100, z5, tool0;
MoveL Offs(p0,30.359199999999998,140.9432, 0), v100, z5, tool0;
MoveL Offs(p0,29.9375,142.5875, 0), v100, z5, tool0;
MoveL Offs(p0,29.596799999999995,144.4568, 0), v100, z5, tool0;
MoveL Offs(p0,29.344899999999996,146.5169, 0), v100, z5, tool0;
MoveL Offs(p0,29.189600000000006,148.73360000000002, 0), v100, z5, tool0;
MoveL Offs(p0,29.1387,151.0727, 0), v100, z5, tool0;
MoveL Offs(p0,29.2,153.5, 0), v100, z5, tool0;
MoveL Offs(p0,29.494400000000006,157.13600000000002, 0), v100, z5, tool0;
MoveL Offs(p0,29.7031,158.702, 0), v100, z5, tool0;
MoveL Offs(p0,29.971200000000003,160.172, 0), v100, z5, tool0;
MoveL Offs(p0,30.3125,161.6, 0), v100, z5, tool0;
MoveL Offs(p0,30.740799999999997,163.04000000000002, 0), v100, z5, tool0;
MoveL Offs(p0,31.2699,164.546, 0), v100, z5, tool0;
MoveL Offs(p0,31.913600000000002,166.17200000000003, 0), v100, z5, tool0;
MoveL Offs(p0,32.6857,167.972, 0), v100, z5, tool0;
MoveL Offs(p0,33.6,170.0, 0), v100, z5, tool0;
MoveL Offs(p0,34.9031,172.64610000000002, 0), v100, z5, tool0;
MoveL Offs(p0,36.320800000000006,175.31680000000003, 0), v100, z5, tool0;
MoveL Offs(p0,37.8057,177.9407, 0), v100, z5, tool0;
MoveL Offs(p0,39.3104,180.44639999999998, 0), v100, z5, tool0;
MoveL Offs(p0,40.7875,182.7625, 0), v100, z5, tool0;
MoveL Offs(p0,42.1896,184.8176, 0), v100, z5, tool0;
MoveL Offs(p0,43.4693,186.5403, 0), v100, z5, tool0;
MoveL Offs(p0,44.5792,187.85920000000002, 0), v100, z5, tool0;
MoveL Offs(p0,45.4719,188.7029, 0), v100, z5, tool0;
MoveL Offs(p0,46.1,189.0, 0), v100, z5, tool0;
MoveL Offs(p0,46.5149,188.72729999999999, 0), v100, z5, tool0;
MoveL Offs(p0,46.632799999999996,188.52960000000002, 0), v100, z5, tool0;
MoveL Offs(p0,46.7375,188.2875, 0), v100, z5, tool0;
MoveL Offs(p0,46.8272,188.0064, 0), v100, z5, tool0;
MoveL Offs(p0,46.900099999999995,187.6917, 0), v100, z5, tool0;
MoveL Offs(p0,46.9544,187.34880000000004, 0), v100, z5, tool0;
MoveL Offs(p0,46.9883,186.98309999999998, 0), v100, z5, tool0;
MoveL Offs(p0,47.0,186.6, 0), v100, z5, tool0;
MoveL Offs(p0,47.0,186.6, 0), v100, z5, tool0;
MoveJ Offs(p0,244.9,183.7, 10), v100, z1, tool0;
MoveL Offs(p0,244.64660000000003,181.67530000000002, 0), v100, z5, tool0;
MoveL Offs(p0,244.54080000000013,179.37040000000007, 0), v100, z5, tool0;
MoveL Offs(p0,244.57419999999996,176.85909999999998, 0), v100, z5, tool0;
MoveL Offs(p0,245.42559999999997,168.8248, 0), v100, z5, tool0;
MoveL Offs(p0,245.93179999999998,166.2259, 0), v100, z5, tool0;
MoveL Offs(p0,246.53519999999997,163.7896, 0), v100, z5, tool0;
MoveL Offs(p0,247.22740000000005,161.58970000000002, 0), v100, z5, tool0;
MoveL Offs(p0,248.0,159.7, 0), v100, z5, tool0;
MoveL Offs(p0,248.39720000000003,158.91100000000003, 0), v100, z5, tool0;
MoveL Offs(p0,248.86160000000004,158.05600000000004, 0), v100, z5, tool0;
MoveL Offs(p0,249.38240000000002,157.15299999999996, 0), v100, z5, tool0;
MoveL Offs(p0,249.94880000000003,156.22000000000003, 0), v100, z5, tool0;
MoveL Offs(p0,250.55,155.275, 0), v100, z5, tool0;
MoveL Offs(p0,251.1752,154.33599999999998, 0), v100, z5, tool0;
MoveL Offs(p0,251.8136,153.421, 0), v100, z5, tool0;
MoveL Offs(p0,252.45440000000002,152.548, 0), v100, z5, tool0;
MoveL Offs(p0,253.08679999999998,151.735, 0), v100, z5, tool0;
MoveL Offs(p0,253.7,151.0, 0), v100, z5, tool0;
MoveL Offs(p0,257.3,146.9, 0), v100, z5, tool0;
MoveL Offs(p0,253.0,142.5, 0), v100, z5, tool0;
MoveL Offs(p0,250.3838,140.0517, 0), v100, z5, tool0;
MoveL Offs(p0,247.5744000000001,137.86560000000003, 0), v100, z5, tool0;
MoveL Offs(p0,244.57059999999996,135.9399, 0), v100, z5, tool0;
MoveL Offs(p0,241.3712,134.27280000000002, 0), v100, z5, tool0;
MoveL Offs(p0,237.975,132.8625, 0), v100, z5, tool0;
MoveL Offs(p0,234.3808,131.7072, 0), v100, z5, tool0;
MoveL Offs(p0,230.58739999999997,130.80509999999998, 0), v100, z5, tool0;
MoveL Offs(p0,226.5936,130.1544, 0), v100, z5, tool0;
MoveL Offs(p0,222.3982,129.7533, 0), v100, z5, tool0;
MoveL Offs(p0,218.0,129.6, 0), v100, z5, tool0;
MoveL Offs(p0,209.49949999999998,130.01579999999998, 0), v100, z5, tool0;
MoveL Offs(p0,207.248,130.3776, 0), v100, z5, tool0;
MoveL Offs(p0,205.2125,130.875, 0), v100, z5, tool0;
MoveL Offs(p0,203.348,131.5224, 0), v100, z5, tool0;
MoveL Offs(p0,201.60949999999997,132.3342, 0), v100, z5, tool0;
MoveL Offs(p0,199.95200000000003,133.3248, 0), v100, z5, tool0;
MoveL Offs(p0,198.33050000000003,134.5086, 0), v100, z5, tool0;
MoveL Offs(p0,196.7,135.9, 0), v100, z5, tool0;
MoveL Offs(p0,195.13690000000003,137.40640000000002, 0), v100, z5, tool0;
MoveL Offs(p0,193.74720000000005,138.98720000000006, 0), v100, z5, tool0;
MoveL Offs(p0,192.53029999999998,140.64479999999998, 0), v100, z5, tool0;
MoveL Offs(p0,191.48560000000003,142.3816, 0), v100, z5, tool0;
MoveL Offs(p0,190.6125,144.2, 0), v100, z5, tool0;
MoveL Offs(p0,189.9104,146.1024, 0), v100, z5, tool0;
MoveL Offs(p0,189.37869999999998,148.0912, 0), v100, z5, tool0;
MoveL Offs(p0,189.01680000000002,150.1688, 0), v100, z5, tool0;
MoveL Offs(p0,188.8241,152.3376, 0), v100, z5, tool0;
MoveL Offs(p0,188.8,154.6, 0), v100, z5, tool0;
MoveL Offs(p0,189.25280000000004,159.18800000000005, 0), v100, z5, tool0;
MoveL Offs(p0,189.7297,161.59750000000003, 0), v100, z5, tool0;
MoveL Offs(p0,190.33440000000002,163.96800000000002, 0), v100, z5, tool0;
MoveL Offs(p0,191.0375,166.2125, 0), v100, z5, tool0;
MoveL Offs(p0,191.8096,168.24399999999997, 0), v100, z5, tool0;
MoveL Offs(p0,192.6213,169.9755, 0), v100, z5, tool0;
MoveL Offs(p0,193.44320000000002,171.32, 0), v100, z5, tool0;
MoveL Offs(p0,194.2459,172.1905, 0), v100, z5, tool0;
MoveL Offs(p0,195.0,172.5, 0), v100, z5, tool0;
MoveL Offs(p0,195.56560000000007,172.28480000000005, 0), v100, z5, tool0;
MoveL Offs(p0,195.90089999999998,172.03019999999998, 0), v100, z5, tool0;
MoveL Offs(p0,196.26080000000002,171.6904, 0), v100, z5, tool0;
MoveL Offs(p0,196.6375,171.275, 0), v100, z5, tool0;
MoveL Offs(p0,197.0232,170.7936, 0), v100, z5, tool0;
MoveL Offs(p0,197.4101,170.2558, 0), v100, z5, tool0;
MoveL Offs(p0,197.7904,169.6712, 0), v100, z5, tool0;
MoveL Offs(p0,198.15630000000002,169.04940000000002, 0), v100, z5, tool0;
MoveL Offs(p0,198.5,168.4, 0), v100, z5, tool0;
MoveL Offs(p0,199.30280000000002,166.8111, 0), v100, z5, tool0;
MoveL Offs(p0,200.09840000000005,165.39680000000004, 0), v100, z5, tool0;
MoveL Offs(p0,200.8976,164.1457, 0), v100, z5, tool0;
MoveL Offs(p0,201.7112,163.0464, 0), v100, z5, tool0;
MoveL Offs(p0,202.55,162.0875, 0), v100, z5, tool0;
MoveL Offs(p0,203.4248,161.2576, 0), v100, z5, tool0;
MoveL Offs(p0,204.3464,160.5453, 0), v100, z5, tool0;
MoveL Offs(p0,205.32560000000004,159.9392, 0), v100, z5, tool0;
MoveL Offs(p0,206.3732,159.4279, 0), v100, z5, tool0;
MoveL Offs(p0,207.5,159.0, 0), v100, z5, tool0;
MoveL Offs(p0,209.21200000000005,158.51450000000003, 0), v100, z5, tool0;
MoveL Offs(p0,210.73200000000006,158.29600000000005, 0), v100, z5, tool0;
MoveL Offs(p0,212.12599999999998,158.4015, 0), v100, z5, tool0;
MoveL Offs(p0,214.8,159.8125, 0), v100, z5, tool0;
MoveL Offs(p0,216.212,161.23200000000003, 0), v100, z5, tool0;
MoveL Offs(p0,217.762,163.2035, 0), v100, z5, tool0;
MoveL Offs(p0,219.516,165.78400000000002, 0), v100, z5, tool0;
MoveL Offs(p0,221.54000000000002,169.03050000000002, 0), v100, z5, tool0;
MoveL Offs(p0,223.9,173.0, 0), v100, z5, tool0;
MoveL Offs(p0,224.70059999999998,174.30970000000005, 0), v100, z5, tool0;
MoveL Offs(p0,225.44480000000004,175.43760000000003, 0), v100, z5, tool0;
MoveL Offs(p0,226.16619999999998,176.4119, 0), v100, z5, tool0;
MoveL Offs(p0,226.89840000000004,177.2608, 0), v100, z5, tool0;
MoveL Offs(p0,227.675,178.0125, 0), v100, z5, tool0;
MoveL Offs(p0,228.52960000000002,178.69519999999997, 0), v100, z5, tool0;
MoveL Offs(p0,229.4958,179.3371, 0), v100, z5, tool0;
MoveL Offs(p0,230.6072,179.96640000000002, 0), v100, z5, tool0;
MoveL Offs(p0,231.8974,180.6113, 0), v100, z5, tool0;
MoveL Offs(p0,233.4,181.3, 0), v100, z5, tool0;
MoveL Offs(p0,234.43780000000007,181.77500000000003, 0), v100, z5, tool0;
MoveL Offs(p0,235.4984000000001,182.2920000000001, 0), v100, z5, tool0;
MoveL Offs(p0,236.56259999999997,182.839, 0), v100, z5, tool0;
MoveL Offs(p0,237.6112,183.40400000000005, 0), v100, z5, tool0;
MoveL Offs(p0,238.625,183.975, 0), v100, z5, tool0;
MoveL Offs(p0,239.5848,184.54, 0), v100, z5, tool0;
MoveL Offs(p0,240.4714,185.087, 0), v100, z5, tool0;
MoveL Offs(p0,241.26560000000003,185.60399999999998, 0), v100, z5, tool0;
MoveL Offs(p0,241.94819999999999,186.079, 0), v100, z5, tool0;
MoveL Offs(p0,242.5,186.5, 0), v100, z5, tool0;
MoveL Offs(p0,243.0,186.87750000000003, 0), v100, z5, tool0;
MoveL Offs(p0,243.47600000000003,187.22800000000007, 0), v100, z5, tool0;
MoveL Offs(p0,243.92199999999997,187.5485, 0), v100, z5, tool0;
MoveL Offs(p0,244.33200000000002,187.836, 0), v100, z5, tool0;
MoveL Offs(p0,244.7,188.0875, 0), v100, z5, tool0;
MoveL Offs(p0,245.01999999999998,188.3, 0), v100, z5, tool0;
MoveL Offs(p0,245.28599999999997,188.4705, 0), v100, z5, tool0;
MoveL Offs(p0,245.49200000000002,188.59600000000003, 0), v100, z5, tool0;
MoveL Offs(p0,245.632,188.67350000000002, 0), v100, z5, tool0;
MoveL Offs(p0,245.7,188.7, 0), v100, z5, tool0;
MoveL Offs(p0,245.4264,186.5976, 0), v100, z5, tool0;
MoveL Offs(p0,245.3122,185.9518, 0), v100, z5, tool0;
MoveL Offs(p0,245.1848,185.24720000000002, 0), v100, z5, tool0;
MoveL Offs(p0,245.04659999999998,184.4934, 0), v100, z5, tool0;
MoveL Offs(p0,244.9,183.7, 0), v100, z5, tool0;
MoveL Offs(p0,244.9,183.7, 0), v100, z5, tool0;
MoveJ Offs(p0,261.9,182.3, 10), v100, z1, tool0;
MoveL Offs(p0,262.2333,180.68970000000002, 0), v100, z5, tool0;
MoveL Offs(p0,262.51440000000014,179.13760000000008, 0), v100, z5, tool0;
MoveL Offs(p0,262.7451,177.6119, 0), v100, z5, tool0;
MoveL Offs(p0,262.92719999999997,176.0808, 0), v100, z5, tool0;
MoveL Offs(p0,263.0625,174.5125, 0), v100, z5, tool0;
MoveL Offs(p0,263.15279999999996,172.8752, 0), v100, z5, tool0;
MoveL Offs(p0,263.19989999999996,171.1371, 0), v100, z5, tool0;
MoveL Offs(p0,263.20560000000006,169.26640000000003, 0), v100, z5, tool0;
MoveL Offs(p0,263.1717,167.2313, 0), v100, z5, tool0;
MoveL Offs(p0,263.1,165.0, 0), v100, z5, tool0;
MoveL Offs(p0,262.9,159.5, 0), v100, z5, tool0;
MoveL Offs(p0,260.5,162.5, 0), v100, z5, tool0;
MoveL Offs(p0,259.28260000000006,164.22430000000003, 0), v100, z5, tool0;
MoveL Offs(p0,258.2728000000001,166.19040000000004, 0), v100, z5, tool0;
MoveL Offs(p0,257.4742,168.35809999999998, 0), v100, z5, tool0;
MoveL Offs(p0,256.89040000000006,170.68720000000002, 0), v100, z5, tool0;
MoveL Offs(p0,256.525,173.1375, 0), v100, z5, tool0;
MoveL Offs(p0,256.3816,175.66879999999998, 0), v100, z5, tool0;
MoveL Offs(p0,256.4638,178.2409, 0), v100, z5, tool0;
MoveL Offs(p0,256.77520000000004,180.81360000000004, 0), v100, z5, tool0;
MoveL Offs(p0,257.3194,183.3467, 0), v100, z5, tool0;
MoveL Offs(p0,258.1,185.8, 0), v100, z5, tool0;
MoveL Offs(p0,258.46290000000005,186.62810000000002, 0), v100, z5, tool0;
MoveL Offs(p0,258.8312000000001,187.19280000000006, 0), v100, z5, tool0;
MoveL Offs(p0,259.2043,187.4947, 0), v100, z5, tool0;
MoveL Offs(p0,259.58160000000004,187.5344, 0), v100, z5, tool0;
MoveL Offs(p0,259.9625,187.3125, 0), v100, z5, tool0;
MoveL Offs(p0,260.3464,186.8296, 0), v100, z5, tool0;
MoveL Offs(p0,260.7327,186.0863, 0), v100, z5, tool0;
MoveL Offs(p0,261.12080000000003,185.0832, 0), v100, z5, tool0;
MoveL Offs(p0,261.5101,183.8209, 0), v100, z5, tool0;
MoveL Offs(p0,261.9,182.3, 0), v100, z5, tool0;
MoveL Offs(p0,261.9,182.3, 0), v100, z5, tool0;
MoveJ Offs(p0,47.7,177.8, 10), v100, z1, tool0;
MoveL Offs(p0,47.4381,177.3689, 0), v100, z5, tool0;
MoveL Offs(p0,47.3592,177.3488, 0), v100, z5, tool0;
MoveL Offs(p0,47.2875,177.3875, 0), v100, z5, tool0;
MoveL Offs(p0,47.2248,177.4832, 0), v100, z5, tool0;
MoveL Offs(p0,47.1087,178.0943, 0), v100, z5, tool0;
MoveL Offs(p0,47.1,178.4, 0), v100, z5, tool0;
MoveL Offs(p0,47.340799999999994,179.80349999999999, 0), v100, z5, tool0;
MoveL Offs(p0,47.4232,179.824, 0), v100, z5, tool0;
MoveL Offs(p0,47.5104,179.7905, 0), v100, z5, tool0;
MoveL Offs(p0,47.6,179.7, 0), v100, z5, tool0;
MoveL Offs(p0,47.8106,179.2896, 0), v100, z5, tool0;
MoveL Offs(p0,47.851200000000006,179.10319999999996, 0), v100, z5, tool0;
MoveL Offs(p0,47.875,178.9, 0), v100, z5, tool0;
MoveL Offs(p0,47.8808,178.6848, 0), v100, z5, tool0;
MoveL Offs(p0,47.8674,178.46240000000003, 0), v100, z5, tool0;
MoveL Offs(p0,47.833600000000004,178.23760000000001, 0), v100, z5, tool0;
MoveL Offs(p0,47.7,177.8, 0), v100, z5, tool0;
MoveJ Offs(p0,176.2,170.3, 10), v100, z1, tool0;
MoveL Offs(p0,176.488,162.3944, 0), v100, z5, tool0;
MoveL Offs(p0,176.662,161.1027, 0), v100, z5, tool0;
MoveL Offs(p0,176.872,159.84880000000004, 0), v100, z5, tool0;
MoveL Offs(p0,177.118,158.6441, 0), v100, z5, tool0;
MoveL Offs(p0,177.4,157.5, 0), v100, z5, tool0;
MoveL Offs(p0,177.8161,155.71910000000003, 0), v100, z5, tool0;
MoveL Offs(p0,178.10080000000008,154.20880000000002, 0), v100, z5, tool0;
MoveL Offs(p0,178.24869999999999,152.9577, 0), v100, z5, tool0;
MoveL Offs(p0,178.25439999999998,151.95440000000002, 0), v100, z5, tool0;
MoveL Offs(p0,178.1125,151.1875, 0), v100, z5, tool0;
MoveL Offs(p0,177.81760000000003,150.6456, 0), v100, z5, tool0;
MoveL Offs(p0,176.74720000000002,150.19120000000004, 0), v100, z5, tool0;
MoveL Offs(p0,175.9609,150.25590000000003, 0), v100, z5, tool0;
MoveL Offs(p0,175.0,150.5, 0), v100, z5, tool0;
MoveL Offs(p0,173.45640000000003,151.39040000000003, 0), v100, z5, tool0;
MoveL Offs(p0,171.81920000000005,152.99120000000002, 0), v100, z5, tool0;
MoveL Offs(p0,170.16879999999998,155.1368, 0), v100, z5, tool0;
MoveL Offs(p0,168.58560000000003,157.66160000000002, 0), v100, z5, tool0;
MoveL Offs(p0,167.15,160.4, 0), v100, z5, tool0;
MoveL Offs(p0,165.9424,163.1864, 0), v100, z5, tool0;
MoveL Offs(p0,165.0432,165.8552, 0), v100, z5, tool0;
MoveL Offs(p0,164.5328,168.2408, 0), v100, z5, tool0;
MoveL Offs(p0,164.4916,170.1776, 0), v100, z5, tool0;
MoveL Offs(p0,165.0,171.5, 0), v100, z5, tool0;
MoveL Offs(p0,165.54240000000001,172.01850000000002, 0), v100, z5, tool0;
MoveL Offs(p0,166.3992,172.64800000000005, 0), v100, z5, tool0;
MoveL Offs(p0,167.4948,173.34949999999998, 0), v100, z5, tool0;
MoveL Offs(p0,168.7536,174.084, 0), v100, z5, tool0;
MoveL Offs(p0,170.1,174.8125, 0), v100, z5, tool0;
MoveL Offs(p0,171.4584,175.496, 0), v100, z5, tool0;
MoveL Offs(p0,172.7532,176.0955, 0), v100, z5, tool0;
MoveL Offs(p0,173.9088,176.57200000000003, 0), v100, z5, tool0;
MoveL Offs(p0,174.8496,176.8865, 0), v100, z5, tool0;
MoveL Offs(p0,175.5,177.0, 0), v100, z5, tool0;
MoveL Offs(p0,175.86080000000004,176.70640000000006, 0), v100, z5, tool0;
MoveL Offs(p0,175.99769999999998,176.3466, 0), v100, z5, tool0;
MoveL Offs(p0,176.10640000000004,175.8512, 0), v100, z5, tool0;
MoveL Offs(p0,176.1875,175.225, 0), v100, z5, tool0;
MoveL Offs(p0,176.2416,174.4728, 0), v100, z5, tool0;
MoveL Offs(p0,176.2693,173.5994, 0), v100, z5, tool0;
MoveL Offs(p0,176.2712,172.60960000000003, 0), v100, z5, tool0;
MoveL Offs(p0,176.24790000000002,171.5082, 0), v100, z5, tool0;
MoveL Offs(p0,176.2,170.3, 0), v100, z5, tool0;
MoveL Offs(p0,176.2,170.3, 0), v100, z5, tool0;
MoveJ Offs(p0,186.0,174.3, 10), v100, z1, tool0;
MoveL Offs(p0,188.09879999999998,174.0354, 0), v100, z5, tool0;
MoveL Offs(p0,188.7056,173.95280000000002, 0), v100, z5, tool0;
MoveL Offs(p0,189.25,173.875, 0), v100, z5, tool0;
MoveL Offs(p0,189.72240000000002,173.8032, 0), v100, z5, tool0;
MoveL Offs(p0,190.1132,173.7386, 0), v100, z5, tool0;
MoveL Offs(p0,190.4128,173.6824, 0), v100, z5, tool0;
MoveL Offs(p0,190.6116,173.6358, 0), v100, z5, tool0;
MoveL Offs(p0,190.7,173.6, 0), v100, z5, tool0;
MoveL Offs(p0,190.4632,172.41440000000003, 0), v100, z5, tool0;
MoveL Offs(p0,190.275,171.8375, 0), v100, z5, tool0;
MoveL Offs(p0,190.04479999999998,171.17360000000002, 0), v100, z5, tool0;
MoveL Offs(p0,189.7774,170.43529999999998, 0), v100, z5, tool0;
MoveL Offs(p0,189.4776,169.63520000000003, 0), v100, z5, tool0;
MoveL Offs(p0,189.15019999999998,168.78590000000003, 0), v100, z5, tool0;
MoveL Offs(p0,188.8,167.9, 0), v100, z5, tool0;
MoveL Offs(p0,187.7607,164.71570000000003, 0), v100, z5, tool0;
MoveL Offs(p0,187.03760000000005,161.33760000000004, 0), v100, z5, tool0;
MoveL Offs(p0,186.6229,157.8479, 0), v100, z5, tool0;
MoveL Offs(p0,186.5088,154.3288, 0), v100, z5, tool0;
MoveL Offs(p0,186.6875,150.8625, 0), v100, z5, tool0;
MoveL Offs(p0,187.15119999999996,147.53119999999998, 0), v100, z5, tool0;
MoveL Offs(p0,187.8921,144.41709999999998, 0), v100, z5, tool0;
MoveL Offs(p0,190.17430000000002,139.1693, 0), v100, z5, tool0;
MoveL Offs(p0,191.7,137.2, 0), v100, z5, tool0;
MoveL Offs(p0,192.33800000000005,136.5312, 0), v100, z5, tool0;
MoveL Offs(p0,192.74800000000005,136.02560000000005, 0), v100, z5, tool0;
MoveL Offs(p0,192.924,135.6844, 0), v100, z5, tool0;
MoveL Offs(p0,192.86000000000004,135.5088, 0), v100, z5, tool0;
MoveL Offs(p0,192.55,135.5, 0), v100, z5, tool0;
MoveL Offs(p0,191.988,135.6592, 0), v100, z5, tool0;
MoveL Offs(p0,191.16799999999998,135.9876, 0), v100, z5, tool0;
MoveL Offs(p0,190.084,136.4864, 0), v100, z5, tool0;
MoveL Offs(p0,187.1,138.0, 0), v100, z5, tool0;
MoveL Offs(p0,184.94290000000004,139.2724, 0), v100, z5, tool0;
MoveL Offs(p0,182.58720000000005,140.84720000000004, 0), v100, z5, tool0;
MoveL Offs(p0,180.17629999999997,142.6008, 0), v100, z5, tool0;
MoveL Offs(p0,177.8536,144.4096, 0), v100, z5, tool0;
MoveL Offs(p0,175.7625,146.15, 0), v100, z5, tool0;
MoveL Offs(p0,174.0464,147.6984, 0), v100, z5, tool0;
MoveL Offs(p0,172.8487,148.9312, 0), v100, z5, tool0;
MoveL Offs(p0,172.3128,149.72480000000002, 0), v100, z5, tool0;
MoveL Offs(p0,172.58210000000003,149.9556, 0), v100, z5, tool0;
MoveL Offs(p0,173.8,149.5, 0), v100, z5, tool0;
MoveL Offs(p0,174.46390000000002,149.19710000000003, 0), v100, z5, tool0;
MoveL Offs(p0,175.07920000000004,148.94880000000003, 0), v100, z5, tool0;
MoveL Offs(p0,175.65130000000002,148.7557, 0), v100, z5, tool0;
MoveL Offs(p0,176.18560000000002,148.6184, 0), v100, z5, tool0;
MoveL Offs(p0,176.6875,148.5375, 0), v100, z5, tool0;
MoveL Offs(p0,177.1624,148.5136, 0), v100, z5, tool0;
MoveL Offs(p0,177.6157,148.5473, 0), v100, z5, tool0;
MoveL Offs(p0,178.05280000000002,148.63920000000002, 0), v100, z5, tool0;
MoveL Offs(p0,178.47910000000002,148.7899, 0), v100, z5, tool0;
MoveL Offs(p0,178.9,149.0, 0), v100, z5, tool0;
MoveL Offs(p0,179.38660000000004,149.26, 0), v100, z5, tool0;
MoveL Offs(p0,179.76880000000003,149.52000000000004, 0), v100, z5, tool0;
MoveL Offs(p0,180.05019999999996,149.81, 0), v100, z5, tool0;
MoveL Offs(p0,180.2344,150.16000000000003, 0), v100, z5, tool0;
MoveL Offs(p0,180.325,150.6, 0), v100, z5, tool0;
MoveL Offs(p0,180.3256,151.16000000000003, 0), v100, z5, tool0;
MoveL Offs(p0,180.2398,151.86999999999998, 0), v100, z5, tool0;
MoveL Offs(p0,180.0712,152.76000000000002, 0), v100, z5, tool0;
MoveL Offs(p0,179.8234,153.85999999999999, 0), v100, z5, tool0;
MoveL Offs(p0,179.5,155.2, 0), v100, z5, tool0;
MoveL Offs(p0,179.29340000000002,156.07350000000002, 0), v100, z5, tool0;
MoveL Offs(p0,179.09520000000006,156.94400000000002, 0), v100, z5, tool0;
MoveL Offs(p0,178.90779999999998,157.79649999999998, 0), v100, z5, tool0;
MoveL Offs(p0,178.73359999999997,158.616, 0), v100, z5, tool0;
MoveL Offs(p0,178.575,159.3875, 0), v100, z5, tool0;
MoveL Offs(p0,178.43439999999998,160.096, 0), v100, z5, tool0;
MoveL Offs(p0,178.31419999999997,160.72650000000002, 0), v100, z5, tool0;
MoveL Offs(p0,178.2168,161.264, 0), v100, z5, tool0;
MoveL Offs(p0,178.14460000000003,161.69350000000003, 0), v100, z5, tool0;
MoveL Offs(p0,178.1,162.0, 0), v100, z5, tool0;
MoveL Offs(p0,177.9,163.8375, 0), v100, z5, tool0;
MoveL Offs(p0,177.8192,164.304, 0), v100, z5, tool0;
MoveL Offs(p0,177.7276,164.78249999999997, 0), v100, z5, tool0;
MoveL Offs(p0,177.62640000000002,165.264, 0), v100, z5, tool0;
MoveL Offs(p0,177.51680000000002,165.7395, 0), v100, z5, tool0;
MoveL Offs(p0,177.4,166.2, 0), v100, z5, tool0;
MoveL Offs(p0,177.18400000000003,168.5248, 0), v100, z5, tool0;
MoveL Offs(p0,177.175,169.2125, 0), v100, z5, tool0;
MoveL Offs(p0,177.18400000000003,169.9152, 0), v100, z5, tool0;
MoveL Offs(p0,177.75520000000006,174.02480000000006, 0), v100, z5, tool0;
MoveL Offs(p0,177.9373,174.55569999999997, 0), v100, z5, tool0;
MoveL Offs(p0,178.12960000000004,174.9744, 0), v100, z5, tool0;
MoveL Offs(p0,178.3375,175.2875, 0), v100, z5, tool0;
MoveL Offs(p0,178.5664,175.5016, 0), v100, z5, tool0;
MoveL Offs(p0,178.82170000000002,175.6233, 0), v100, z5, tool0;
MoveL Offs(p0,179.10880000000003,175.6592, 0), v100, z5, tool0;
MoveL Offs(p0,179.43310000000002,175.6159, 0), v100, z5, tool0;
MoveL Offs(p0,179.8,175.5, 0), v100, z5, tool0;
MoveL Offs(p0,180.55040000000005,175.25040000000004, 0), v100, z5, tool0;
MoveL Offs(p0,181.0636,175.1211, 0), v100, z5, tool0;
MoveL Offs(p0,181.65120000000002,174.99120000000002, 0), v100, z5, tool0;
MoveL Offs(p0,182.3,174.8625, 0), v100, z5, tool0;
MoveL Offs(p0,182.99679999999998,174.7368, 0), v100, z5, tool0;
MoveL Offs(p0,183.72840000000002,174.6159, 0), v100, z5, tool0;
MoveL Offs(p0,184.48160000000001,174.5016, 0), v100, z5, tool0;
MoveL Offs(p0,185.24320000000003,174.3957, 0), v100, z5, tool0;
MoveL Offs(p0,186.0,174.3, 0), v100, z5, tool0;
MoveL Offs(p0,186.0,174.3, 0), v100, z5, tool0;
MoveJ Offs(p0,164.0,164.5, 10), v100, z1, tool0;
MoveL Offs(p0,163.792,164.22960000000003, 0), v100, z5, tool0;
MoveL Offs(p0,163.6875,164.2625, 0), v100, z5, tool0;
MoveL Offs(p0,163.14950000000002,164.7781, 0), v100, z5, tool0;
MoveL Offs(p0,163.0,165.0, 0), v100, z5, tool0;
MoveL Offs(p0,162.70400000000004,165.51920000000004, 0), v100, z5, tool0;
MoveL Offs(p0,162.5635,165.79829999999998, 0), v100, z5, tool0;
MoveL Offs(p0,162.432,166.0816, 0), v100, z5, tool0;
MoveL Offs(p0,162.3125,166.3625, 0), v100, z5, tool0;
MoveL Offs(p0,162.208,166.6344, 0), v100, z5, tool0;
MoveL Offs(p0,162.1215,166.89069999999998, 0), v100, z5, tool0;
MoveL Offs(p0,162.056,167.1248, 0), v100, z5, tool0;
MoveL Offs(p0,162.01450000000003,167.3301, 0), v100, z5, tool0;
MoveL Offs(p0,162.0,167.5, 0), v100, z5, tool0;
MoveL Offs(p0,162.208,167.81360000000004, 0), v100, z5, tool0;
MoveL Offs(p0,162.3125,167.775, 0), v100, z5, tool0;
MoveL Offs(p0,162.8505,167.2246, 0), v100, z5, tool0;
MoveL Offs(p0,163.0,167.0, 0), v100, z5, tool0;
MoveL Offs(p0,163.29600000000002,166.49040000000008, 0), v100, z5, tool0;
MoveL Offs(p0,163.4365,166.2206, 0), v100, z5, tool0;
MoveL Offs(p0,163.56800000000004,165.9472, 0), v100, z5, tool0;
MoveL Offs(p0,163.6875,165.675, 0), v100, z5, tool0;
MoveL Offs(p0,163.792,165.40879999999999, 0), v100, z5, tool0;
MoveL Offs(p0,163.87849999999997,165.1534, 0), v100, z5, tool0;
MoveL Offs(p0,163.94400000000002,164.91360000000003, 0), v100, z5, tool0;
MoveL Offs(p0,163.9855,164.6942, 0), v100, z5, tool0;
MoveL Offs(p0,164.0,164.5, 0), v100, z5, tool0;
MoveL Offs(p0,164.0,164.5, 0), v100, z5, tool0;
MoveJ Offs(p0,28.3,162.8, 10), v100, z1, tool0;
MoveL Offs(p0,28.051299999999998,161.3719, 0), v100, z5, tool0;
MoveL Offs(p0,27.84640000000001,159.34320000000005, 0), v100, z5, tool0;
MoveL Offs(p0,27.687099999999997,156.85729999999998, 0), v100, z5, tool0;
MoveL Offs(p0,27.575200000000002,154.0576, 0), v100, z5, tool0;
MoveL Offs(p0,27.5125,151.0875, 0), v100, z5, tool0;
MoveL Offs(p0,27.500799999999998,148.0904, 0), v100, z5, tool0;
MoveL Offs(p0,27.5419,145.2097, 0), v100, z5, tool0;
MoveL Offs(p0,27.637600000000003,142.5888, 0), v100, z5, tool0;
MoveL Offs(p0,27.789700000000003,140.3711, 0), v100, z5, tool0;
MoveL Offs(p0,28.0,138.7, 0), v100, z5, tool0;
MoveL Offs(p0,27.55,135.9875, 0), v100, z5, tool0;
MoveL Offs(p0,27.020799999999998,135.5752, 0), v100, z5, tool0;
MoveL Offs(p0,26.286399999999997,135.1461, 0), v100, z5, tool0;
MoveL Offs(p0,25.3216,134.67440000000002, 0), v100, z5, tool0;
MoveL Offs(p0,24.1012,134.1343, 0), v100, z5, tool0;
MoveL Offs(p0,22.6,133.5, 0), v100, z5, tool0;
MoveL Offs(p0,21.630000000000003,133.11980000000003, 0), v100, z5, tool0;
MoveL Offs(p0,20.708000000000006,132.7624, 0), v100, z5, tool0;
MoveL Offs(p0,19.845999999999997,132.4326, 0), v100, z5, tool0;
MoveL Offs(p0,19.056,132.1352, 0), v100, z5, tool0;
MoveL Offs(p0,18.35,131.875, 0), v100, z5, tool0;
MoveL Offs(p0,17.740000000000002,131.6568, 0), v100, z5, tool0;
MoveL Offs(p0,17.238,131.4854, 0), v100, z5, tool0;
MoveL Offs(p0,16.856,131.3656, 0), v100, z5, tool0;
MoveL Offs(p0,16.606,131.30220000000003, 0), v100, z5, tool0;
MoveL Offs(p0,16.5,131.3, 0), v100, z5, tool0;
